C03638=1020.373,204.181,377.085,168.836,50.366,159.543
C03639=1020.379,204.400,377.063,168.838,50.360,159.542
C03640=1020.384,204.618,377.040,168.842,50.355,159.542
C03641=1020.390,204.838,377.018,168.844,50.349,159.541
C03642=1020.396,205.057,376.996,168.848,50.344,159.540
C03643=1020.401,205.276,376.974,168.852,50.339,159.540
C03644=1020.406,205.494,376.951,168.855,50.333,159.539
C03645=1020.412,205.713,376.930,168.858,50.328,159.539
C03646=1020.418,205.961,376.904,168.861,50.322,159.538
C03647=1020.424,206.210,376.879,168.864,50.316,159.537
C03648=1020.431,206.459,376.854,168.868,50.310,159.536
C03649=1020.437,206.707,376.828,168.872,50.304,159.536
C03650=1020.443,206.956,376.803,168.876,50.298,159.535
C03651=1020.449,207.204,376.778,168.879,50.292,159.535
C03652=1020.455,207.453,376.753,168.882,50.287,159.534
C03653=1020.461,207.701,376.727,168.886,50.281,159.533
C03654=1020.466,207.950,376.701,168.890,50.275,159.532
C03655=1020.473,208.198,376.675,168.894,50.269,159.532
C03656=1020.479,208.447,376.650,168.897,50.263,159.531
C03657=1020.485,208.696,376.625,168.900,50.257,159.530
C03658=1020.492,208.944,376.599,168.904,50.251,159.530
C03659=1020.498,209.193,376.574,168.908,50.245,159.529
C03660=1020.504,209.442,376.549,168.912,50.239,159.528
C03661=1020.510,209.690,376.523,168.914,50.233,159.528
C03662=1020.516,209.939,376.497,168.919,50.228,159.527
C03663=1020.522,210.187,376.471,168.922,50.222,159.527
C03664=1020.528,210.436,376.446,168.926,50.216,159.526
C03665=1020.535,210.685,376.421,168.929,50.210,159.525
C03666=1020.540,210.933,376.394,168.933,50.205,159.525
C03667=1020.547,211.182,376.369,168.937,50.199,159.524
C03668=1020.553,211.431,376.343,168.941,50.193,159.524
C03669=1020.559,211.680,376.317,168.944,50.187,159.523
C03670=1020.565,211.928,376.291,168.948,50.182,159.522
C03671=1020.572,212.177,376.266,168.952,50.176,159.522
C03672=1020.577,212.426,376.240,168.954,50.170,159.521
C03673=1020.584,212.674,376.214,168.958,50.164,159.520
C03674=1020.590,212.923,376.188,168.962,50.159,159.520
C03675=1020.596,213.171,376.163,168.966,50.153,159.519
C03676=1020.602,213.420,376.136,168.969,50.147,159.518
C03677=1020.608,213.668,376.111,168.973,50.142,159.518
C03678=1020.614,213.916,376.085,168.977,50.136,159.517
C03679=1020.620,214.165,376.059,168.980,50.130,159.517
C03680=1020.626,214.414,376.034,168.984,50.125,159.516
C03681=1020.633,214.663,376.007,168.988,50.119,159.515
C03682=1020.639,214.912,375.981,168.992,50.114,159.515
C03683=1020.645,215.160,375.955,168.995,50.108,159.514
C03684=1020.651,215.408,375.930,168.999,50.102,159.514
C03685=1020.657,215.657,375.903,169.003,50.097,159.513
C03686=1020.663,215.905,375.878,169.006,50.091,159.512
C03687=1020.670,216.154,375.853,169.010,50.086,159.512
C03688=1020.676,216.403,375.826,169.014,50.080,159.511
C03689=1020.682,216.652,375.800,169.017,50.074,159.511
C03690=1020.689,216.900,375.774,169.021,50.069,159.510
C03691=1020.694,217.149,375.748,169.025,50.063,159.509
C03692=1020.701,217.397,375.722,169.029,50.058,159.509
C03693=1020.707,217.646,375.697,169.032,50.052,159.508
C03694=1020.714,217.894,375.670,169.036,50.047,159.508
C03695=1020.720,218.143,375.644,169.040,50.041,159.507
C03696=1020.726,218.391,375.618,169.044,50.035,159.507
C03697=1020.732,218.640,375.592,169.047,50.030,159.506
C03698=1020.737,218.861,375.569,169.050,50.025,159.506
C03699=1020.743,219.082,375.545,169.053,50.020,159.505
C03700=1020.748,219.304,375.522,169.057,50.015,159.505
C03701=1020.754,219.525,375.498,169.060,50.011,159.504
C03702=1020.759,219.747,375.475,169.063,50.006,159.504
C03703=1020.764,219.968,375.451,169.066,50.001,159.503
C03704=1020.770,220.190,375.429,169.070,49.996,159.503
C03705=1020.775,220.410,375.405,169.073,49.991,159.502
C03706=1020.781,220.659,375.378,169.077,49.986,159.502
C03707=1020.788,220.908,375.353,169.081,49.981,159.501
C03708=1020.794,221.157,375.326,169.084,49.976,159.501
C03709=1020.800,221.405,375.299,169.088,49.970,159.500
C03710=1020.806,221.653,375.273,169.092,49.965,159.499
C03711=1020.812,221.902,375.246,169.096,49.960,159.499
C03712=1020.819,222.151,375.221,169.100,49.954,159.498
C03713=1020.824,222.399,375.194,169.103,49.949,159.498
C03714=1020.830,222.647,375.168,169.107,49.943,159.497
C03715=1020.837,222.896,375.141,169.111,49.938,159.497
C03716=1020.843,223.144,375.115,169.114,49.933,159.496
C03717=1020.849,223.393,375.088,169.118,49.927,159.496
C03718=1020.856,223.642,375.062,169.121,49.922,159.495
C03719=1020.861,223.891,375.036,169.126,49.917,159.495
C03720=1020.868,224.139,375.009,169.130,49.912,159.494
C03721=1020.874,224.387,374.983,169.133,49.907,159.494
C03722=1020.880,224.636,374.956,169.137,49.901,159.493
C03723=1020.887,224.884,374.930,169.141,49.895,159.492
C03724=1020.892,225.132,374.903,169.144,49.890,159.492
C03725=1020.899,225.382,374.876,169.149,49.885,159.491
C03726=1020.905,225.630,374.850,169.152,49.880,159.491
C03727=1020.912,225.879,374.823,169.156,49.875,159.490
C03728=1020.918,226.127,374.797,169.160,49.870,159.490
C03729=1020.924,226.375,374.770,169.163,49.865,159.489
C03730=1020.930,226.624,374.743,169.167,49.859,159.489
C03731=1020.937,226.872,374.717,169.171,49.853,159.488
C03732=1020.943,227.120,374.691,169.175,49.849,159.488
C03733=1020.949,227.370,374.664,169.179,49.844,159.488
C03734=1020.955,227.618,374.637,169.182,49.839,159.487
C03735=1020.961,227.866,374.610,169.187,49.834,159.487
C03736=1020.967,228.115,374.583,169.190,49.829,159.486
C03737=1020.973,228.364,374.557,169.194,49.824,159.486
C03738=1020.980,228.612,374.530,169.197,49.819,159.485
C03739=1020.986,228.860,374.503,169.202,49.813,159.485
C03740=1020.992,229.109,374.476,169.206,49.808,159.484
C03741=1020.998,229.358,374.449,169.209,49.803,159.483
C03742=1021.004,229.606,374.423,169.213,49.798,159.483
C03743=1021.010,229.855,374.396,169.216,49.793,159.482
C03744=1021.016,230.103,374.368,169.221,49.788,159.482
C03745=1021.022,230.351,374.342,169.224,49.783,159.482
C03746=1021.028,230.600,374.315,169.228,49.778,159.481
C03747=1021.034,230.848,374.287,169.232,49.773,159.481
C03748=1021.041,231.097,374.260,169.236,49.768,159.480
C03749=1021.047,231.345,374.233,169.241,49.763,159.480
C03750=1021.053,231.594,374.206,169.244,49.758,159.479
C03751=1021.059,231.842,374.179,169.248,49.753,159.479
C03752=1021.065,232.091,374.152,169.251,49.748,159.478
C03753=1021.072,232.339,374.125,169.256,49.744,159.478
C03754=1021.077,232.587,374.098,169.259,49.739,159.478
C03755=1021.084,232.836,374.071,169.263,49.733,159.477
C03756=1021.090,233.084,374.044,169.266,49.728,159.477
C03757=1021.096,233.333,374.017,169.271,49.724,159.476
C03758=1021.101,233.550,373.993,169.275,49.720,159.476
C03759=1021.107,233.767,373.969,169.277,49.716,159.476
C03760=1021.113,233.985,373.945,169.280,49.711,159.475
C03761=1021.117,234.202,373.922,169.284,49.706,159.475
C03762=1021.123,234.419,373.897,169.288,49.702,159.474
C03763=1021.129,234.637,373.874,169.291,49.698,159.474
C03764=1021.134,234.854,373.851,169.295,49.694,159.474
C03765=1021.140,235.071,373.826,169.297,49.690,159.473
C03766=1021.145,235.320,373.800,169.302,49.684,159.473
C03767=1021.152,235.568,373.772,169.306,49.680,159.472
C03768=1021.158,235.817,373.745,169.309,49.675,159.472
C03769=1021.164,236.065,373.717,169.314,49.670,159.472
C03770=1021.171,236.314,373.690,169.317,49.665,159.471
C03771=1021.177,236.562,373.663,169.322,49.661,159.471
C03772=1021.183,236.811,373.636,169.325,49.656,159.470
C03773=1021.189,237.059,373.609,169.329,49.651,159.470
C03774=1021.195,237.307,373.580,169.333,49.646,159.469
C03775=1021.202,237.556,373.553,169.337,49.641,159.469
C03776=1021.208,237.804,373.526,169.341,49.637,159.469
C03777=1021.214,238.053,373.499,169.345,49.632,159.468
C03778=1021.220,238.301,373.472,169.349,49.627,159.468
C03779=1021.227,238.549,373.444,169.353,49.622,159.467
C03780=1021.233,238.798,373.417,169.356,49.618,159.467
C03781=1021.239,239.046,373.389,169.361,49.613,159.466
C03782=1021.246,239.295,373.362,169.364,49.609,159.466
C03783=1021.251,239.543,373.334,169.369,49.604,159.466
C03784=1021.258,239.792,373.307,169.372,49.599,159.465
C03785=1021.264,240.040,373.278,169.377,49.594,159.465
C03786=1021.270,240.288,373.251,169.380,49.590,159.465
C03787=1021.276,240.537,373.223,169.385,49.585,159.464
C03788=1021.282,240.785,373.195,169.388,49.581,159.464
C03789=1021.289,241.033,373.168,169.393,49.576,159.464
C03790=1021.295,241.282,373.141,169.396,49.571,159.463
C03791=1021.301,241.531,373.112,169.400,49.567,159.463
C03792=1021.307,241.779,373.085,169.404,49.562,159.462
C03793=1021.313,242.027,373.057,169.408,49.558,159.462
C03794=1021.320,242.276,373.029,169.412,49.553,159.462
C03795=1021.326,242.524,373.002,169.416,49.549,159.461
C03796=1021.332,242.772,372.973,169.420,49.544,159.461
C03797=1021.338,243.021,372.945,169.424,49.540,159.461
C03798=1021.344,243.268,372.918,169.429,49.535,159.460
C03799=1021.350,243.517,372.890,169.432,49.530,159.460
C03800=1021.357,243.766,372.862,169.436,49.526,159.460
C03801=1021.362,244.014,372.834,169.440,49.522,159.459
C03802=1021.368,244.262,372.806,169.444,49.517,159.459
C03803=1021.375,244.511,372.778,169.448,49.513,159.459
C03804=1021.381,244.760,372.750,169.452,49.509,159.458
C03805=1021.386,245.008,372.722,169.456,49.504,159.458
C03806=1021.393,245.256,372.693,169.460,49.500,159.458
C03807=1021.399,245.504,372.665,169.464,49.496,159.457
C03808=1021.404,245.752,372.637,169.468,49.491,159.457
C03809=1021.411,246.001,372.609,169.472,49.487,159.457
C03810=1021.417,246.250,372.581,169.477,49.482,159.456
C03811=1021.423,246.498,372.552,169.480,49.478,159.456
C03812=1021.429,246.745,372.525,169.485,49.473,159.456
C03813=1021.435,246.994,372.496,169.488,49.469,159.455
C03814=1021.441,247.243,372.468,169.492,49.465,159.455
C03815=1021.448,247.491,372.439,169.497,49.460,159.455
C03816=1021.454,247.740,372.411,169.500,49.456,159.454
C03817=1021.460,247.988,372.383,169.505,49.452,159.454
C03818=1021.465,248.202,372.359,169.508,49.448,159.454
C03819=1021.470,248.416,372.335,169.511,49.444,159.453
C03820=1021.476,248.630,372.310,169.515,49.441,159.453
C03821=1021.482,248.844,372.286,169.518,49.437,159.453
C03822=1021.486,249.058,372.261,169.522,49.433,159.453
C03823=1021.492,249.273,372.237,169.526,49.430,159.452
C03824=1021.497,249.487,372.213,169.529,49.426,159.452
C03825=1021.503,249.701,372.188,169.532,49.422,159.452
C03826=1021.509,249.950,372.160,169.536,49.419,159.452
C03827=1021.515,250.197,372.131,169.541,49.414,159.451
C03828=1021.521,250.445,372.103,169.545,49.410,159.451
C03829=1021.527,250.694,372.075,169.549,49.405,159.451
C03830=1021.533,250.942,372.046,169.553,49.401,159.450
C03831=1021.540,251.191,372.018,169.558,49.396,159.450
C03832=1021.546,251.439,371.989,169.562,49.393,159.450
C03833=1021.552,251.688,371.961,169.565,49.389,159.450
C03834=1021.559,251.936,371.933,169.570,49.384,159.449
C03835=1021.565,252.184,371.904,169.573,49.380,159.449
C03836=1021.571,252.433,371.876,169.578,49.375,159.449
C03837=1021.578,252.680,371.848,169.582,49.372,159.449
C03838=1021.584,252.929,371.819,169.587,49.367,159.448
C03839=1021.590,253.177,371.790,169.590,49.363,159.448
C03840=1021.596,253.425,371.763,169.594,49.359,159.448
C03841=1021.603,253.674,371.733,169.599,49.355,159.447
C03842=1021.609,253.922,371.705,169.602,49.351,159.447
C03843=1021.616,254.170,371.677,169.607,49.346,159.447
C03844=1021.622,254.418,371.648,169.611,49.343,159.447
C03845=1021.628,254.667,371.619,169.616,49.338,159.446
C03846=1021.634,254.915,371.590,169.619,49.334,159.446
C03847=1021.641,255.164,371.563,169.624,49.329,159.446
C03848=1021.647,255.412,371.534,169.628,49.326,159.446
C03849=1021.653,255.660,371.504,169.631,49.322,159.445
C03850=1021.660,255.908,371.477,169.636,49.318,159.445
C03851=1021.666,256.156,371.448,169.640,49.314,159.445
C03852=1021.672,256.405,371.419,169.645,49.309,159.444
C03853=1021.679,256.653,371.391,169.649,49.306,159.444
C03854=1021.685,256.901,371.362,169.653,49.301,159.444
C03855=1021.692,257.151,371.333,169.657,49.297,159.444
C03856=1021.699,257.398,371.305,169.662,49.293,159.444
C03857=1021.705,257.647,371.276,169.666,49.289,159.443
C03858=1021.711,257.895,371.247,169.670,49.285,159.443
C03859=1021.717,258.143,371.218,169.674,49.281,159.443
C03860=1021.724,258.391,371.190,169.678,49.277,159.443
C03861=1021.731,258.639,371.161,169.683,49.273,159.442
C03862=1021.737,258.887,371.132,169.687,49.269,159.442
C03863=1021.744,259.136,371.104,169.691,49.265,159.442
C03864=1021.750,259.384,371.075,169.695,49.260,159.442
C03865=1021.757,259.633,371.046,169.700,49.256,159.441
C03866=1021.764,259.881,371.017,169.704,49.252,159.441
C03867=1021.770,260.129,370.988,169.709,49.248,159.441
C03868=1021.776,260.377,370.959,169.713,49.245,159.441
C03869=1021.782,260.625,370.930,169.716,49.241,159.440
C03870=1021.789,260.873,370.901,169.721,49.237,159.440
C03871=1021.795,261.121,370.872,169.725,49.233,159.440
C03872=1021.801,261.369,370.843,169.730,49.229,159.440
C03873=1021.807,261.618,370.814,169.734,49.225,159.440
C03874=1021.813,261.867,370.784,169.738,49.222,159.440
C03875=1021.820,262.115,370.755,169.743,49.218,159.439
C03876=1021.826,262.363,370.726,169.746,49.214,159.439
C03877=1021.832,262.611,370.697,169.750,49.210,159.439
C03878=1021.838,262.824,370.672,169.754,49.207,159.439
C03879=1021.843,263.038,370.646,169.759,49.204,159.439
C03880=1021.849,263.251,370.621,169.762,49.200,159.439
C03881=1021.854,263.464,370.596,169.766,49.197,159.438
C03882=1021.860,263.678,370.571,169.770,49.193,159.438
C03883=1021.865,263.891,370.546,169.773,49.191,159.438
C03884=1021.870,264.104,370.521,169.777,49.187,159.438
C03885=1021.876,264.318,370.495,169.781,49.184,159.438
C03886=1021.882,264.566,370.466,169.785,49.180,159.438
C03887=1021.888,264.814,370.437,169.789,49.177,159.437
C03888=1021.895,265.062,370.407,169.794,49.173,159.437
C03889=1021.901,265.310,370.378,169.798,49.169,159.437
C03890=1021.908,265.559,370.348,169.803,49.165,159.437
C03891=1021.914,265.807,370.319,169.807,49.162,159.437
C03892=1021.920,266.055,370.289,169.810,49.158,159.437
C03893=1021.926,266.303,370.260,169.815,49.154,159.436
C03894=1021.933,266.552,370.231,169.819,49.150,159.436
C03895=1021.940,266.799,370.201,169.823,49.147,159.436
C03896=1021.945,267.048,370.171,169.828,49.143,159.436
C03897=1021.952,267.296,370.141,169.832,49.139,159.436
C03898=1021.958,267.544,370.112,169.837,49.136,159.436
C03899=1021.965,267.792,370.083,169.841,49.132,159.436
C03900=1021.971,268.040,370.053,169.846,49.129,159.436
C03901=1021.977,268.289,370.023,169.851,49.125,159.435
C03902=1021.984,268.536,369.993,169.855,49.122,159.435
C03903=1021.989,268.785,369.964,169.860,49.118,159.435
C03904=1021.997,269.033,369.934,169.864,49.114,159.435
C03905=1022.003,269.281,369.905,169.868,49.111,159.435
C03906=1022.009,269.528,369.875,169.873,49.107,159.435
C03907=1022.016,269.778,369.845,169.877,49.104,159.435
C03908=1022.022,270.025,369.815,169.882,49.100,159.434
C03909=1022.028,270.273,369.785,169.886,49.097,159.435
C03910=1022.035,270.522,369.755,169.890,49.093,159.434
C03911=1022.041,270.770,369.725,169.895,49.089,159.434
C03912=1022.047,271.017,369.695,169.899,49.086,159.434
C03913=1022.054,271.266,369.666,169.903,49.082,159.434
C03914=1022.060,271.514,369.635,169.908,49.079,159.434
C03915=1022.067,271.762,369.605,169.912,49.076,159.434
C03916=1022.072,272.010,369.576,169.917,49.072,159.434
C03917=1022.079,272.258,369.546,169.921,49.068,159.434
C03918=1022.085,272.506,369.515,169.926,49.066,159.434
C03919=1022.092,272.754,369.486,169.931,49.062,159.433
C03920=1022.098,273.003,369.456,169.935,49.058,159.433
C03921=1022.105,273.251,369.426,169.939,49.055,159.433
C03922=1022.110,273.498,369.395,169.944,49.051,159.433
C03923=1022.118,273.747,369.365,169.948,49.048,159.433
C03924=1022.123,273.995,369.335,169.953,49.045,159.433
C03925=1022.131,274.243,369.305,169.957,49.041,159.433
C03926=1022.136,274.491,369.275,169.961,49.038,159.433
C03927=1022.143,274.739,369.245,169.967,49.035,159.433
C03928=1022.149,274.987,369.215,169.971,49.031,159.433
C03929=1022.156,275.236,369.184,169.975,49.028,159.433
C03930=1022.162,275.483,369.154,169.980,49.024,159.433
C03931=1022.169,275.732,369.124,169.984,49.021,159.433
C03932=1022.175,275.979,369.094,169.989,49.018,159.433
C03933=1022.181,276.228,369.063,169.993,49.014,159.432
C03934=1022.188,276.475,369.033,169.998,49.011,159.432
C03935=1022.194,276.724,369.003,170.003,49.007,159.432
C03936=1022.201,276.971,368.973,170.007,49.005,159.432
C03937=1022.207,277.220,368.942,170.012,49.001,159.432
C03938=1022.213,277.435,368.915,170.015,48.998,159.432
C03939=1022.218,277.651,368.889,170.020,48.995,159.432
C03940=1022.223,277.867,368.862,170.024,48.993,159.432
C03941=1022.230,278.082,368.836,170.027,48.990,159.432
C03942=1022.235,278.298,368.809,170.032,48.987,159.432
C03943=1022.240,278.514,368.783,170.036,48.984,159.432
C03944=1022.245,278.729,368.756,170.039,48.982,159.432
C03945=1022.251,278.945,368.729,170.044,48.979,159.432
C03946=1022.258,279.192,368.699,170.048,48.976,159.432
C03947=1022.264,279.440,368.668,170.053,48.972,159.432
C03948=1022.271,279.689,368.638,170.057,48.969,159.432
C03949=1022.277,279.937,368.607,170.062,48.966,159.432
C03950=1022.283,280.185,368.576,170.067,48.963,159.432
C03951=1022.290,280.432,368.546,170.071,48.960,159.432
C03952=1022.296,280.681,368.515,170.076,48.957,159.432
C03953=1022.303,280.929,368.485,170.081,48.954,159.432
C03954=1022.309,281.176,368.453,170.085,48.951,159.432
C03955=1022.315,281.425,368.423,170.090,48.947,159.432
C03956=1022.322,281.673,368.393,170.094,48.944,159.432
C03957=1022.328,281.920,368.362,170.099,48.941,159.432
C03958=1022.335,282.169,368.331,170.104,48.938,159.432
C03959=1022.342,282.417,368.299,170.108,48.935,159.432
C03960=1022.347,282.665,368.269,170.113,48.932,159.432
C03961=1022.355,282.913,368.239,170.118,48.929,159.432
C03962=1022.361,283.161,368.208,170.122,48.926,159.432
C03963=1022.368,283.409,368.177,170.127,48.923,159.432
C03964=1022.374,283.656,368.146,170.132,48.920,159.432
C03965=1022.380,283.905,368.115,170.137,48.917,159.432
C03966=1022.387,284.153,368.084,170.141,48.913,159.432
C03967=1022.394,284.400,368.054,170.146,48.910,159.432
C03968=1022.400,284.648,368.022,170.151,48.907,159.432
C03969=1022.407,284.897,367.992,170.155,48.904,159.432
C03970=1022.413,285.145,367.960,170.161,48.901,159.432
C03971=1022.420,285.393,367.929,170.165,48.898,159.432
C03972=1022.426,285.640,367.898,170.170,48.895,159.432
C03973=1022.433,285.888,367.867,170.175,48.892,159.432
C03974=1022.439,286.136,367.836,170.179,48.889,159.432
C03975=1022.446,286.385,367.805,170.184,48.886,159.432
C03976=1022.452,286.632,367.774,170.189,48.883,159.432
C03977=1022.459,286.880,367.742,170.194,48.880,159.432
C03978=1022.465,287.128,367.712,170.199,48.878,159.433
C03979=1022.472,287.376,367.680,170.203,48.875,159.433
C03980=1022.479,287.624,367.649,170.208,48.872,159.433
C03981=1022.485,287.871,367.618,170.213,48.869,159.433
C03982=1022.491,288.119,367.586,170.218,48.866,159.433
C03983=1022.498,288.368,367.556,170.222,48.863,159.433
C03984=1022.505,288.616,367.524,170.227,48.860,159.433
C03985=1022.511,288.864,367.492,170.232,48.858,159.433
C03986=1022.517,289.112,367.461,170.237,48.855,159.433
C03987=1022.524,289.360,367.429,170.242,48.852,159.433
C03988=1022.530,289.607,367.398,170.246,48.849,159.433
C03989=1022.537,289.855,367.367,170.251,48.846,159.433
C03990=1022.544,290.103,367.335,170.257,48.844,159.433
C03991=1022.550,290.351,367.304,170.261,48.841,159.433
C03992=1022.557,290.599,367.272,170.266,48.838,159.434
C03993=1022.563,290.847,367.240,170.271,48.835,159.434
C03994=1022.570,291.095,367.209,170.276,48.832,159.434
C03995=1022.576,291.343,367.178,170.281,48.829,159.434
C03996=1022.583,291.591,367.146,170.285,48.827,159.434
C03997=1022.590,291.838,367.115,170.291,48.824,159.434
C03998=1022.595,292.060,367.086,170.295,48.821,159.434
C03999=1022.601,292.281,367.058,170.299,48.819,159.434
C04000=1022.607,292.504,367.029,170.303,48.817,159.434
C04001=1022.614,292.725,367.001,170.308,48.814,159.434
C04002=1022.619,292.947,366.973,170.312,48.812,159.435
C04003=1022.625,293.168,366.945,170.317,48.809,159.435
C04004=1022.631,293.390,366.916,170.321,48.807,159.435
C04005=1022.637,293.613,366.888,170.326,48.805,159.435
C04006=1022.643,293.860,366.856,170.330,48.802,159.435
C04007=1022.649,294.109,366.824,170.335,48.800,159.435
C04008=1022.656,294.356,366.792,170.341,48.797,159.435
C04009=1022.662,294.604,366.760,170.345,48.795,159.435
C04010=1022.669,294.852,366.728,170.350,48.792,159.436
C04011=1022.675,295.100,366.695,170.355,48.789,159.436
C04012=1022.681,295.348,366.663,170.360,48.787,159.436
C04013=1022.688,295.595,366.631,170.366,48.785,159.436
C04014=1022.694,295.843,366.599,170.370,48.782,159.436
C04015=1022.701,296.090,366.567,170.375,48.780,159.436
C04016=1022.707,296.339,366.535,170.380,48.777,159.437
C04017=1022.714,296.586,366.502,170.385,48.774,159.437
C04018=1022.720,296.834,366.471,170.390,48.772,159.437
C04019=1022.727,297.082,366.438,170.395,48.769,159.437
C04020=1022.733,297.330,366.407,170.400,48.767,159.437
C04021=1022.740,297.577,366.374,170.405,48.764,159.437
C04022=1022.746,297.825,366.341,170.410,48.762,159.438
C04023=1022.753,298.073,366.310,170.416,48.759,159.438
C04024=1022.759,298.320,366.277,170.420,48.757,159.438
C04025=1022.766,298.569,366.245,170.425,48.754,159.438
C04026=1022.773,298.817,366.212,170.430,48.752,159.438
C04027=1022.779,299.064,366.180,170.435,48.750,159.439
C04028=1022.786,299.312,366.148,170.441,48.747,159.439
C04029=1022.792,299.560,366.116,170.445,48.745,159.439
C04030=1022.799,299.807,366.083,170.451,48.743,159.439
C04031=1022.805,300.055,366.051,170.456,48.740,159.440
C04032=1022.812,300.303,366.018,170.461,48.737,159.440
C04033=1022.819,300.551,365.986,170.466,48.735,159.440
C04034=1022.825,300.798,365.953,170.470,48.733,159.440
C04035=1022.832,301.046,365.921,170.476,48.730,159.440
C04036=1022.839,301.295,365.889,170.481,48.728,159.440
C04037=1022.845,301.542,365.856,170.487,48.726,159.441
C04038=1022.852,301.789,365.824,170.491,48.724,159.441
C04039=1022.858,302.037,365.791,170.497,48.721,159.441
C04040=1022.865,302.285,365.758,170.502,48.719,159.441
C04041=1022.872,302.533,365.726,170.507,48.716,159.442
C04042=1022.879,302.780,365.693,170.512,48.714,159.442
C04043=1022.886,303.027,365.661,170.518,48.712,159.442
C04044=1022.892,303.276,365.629,170.522,48.709,159.442
C04045=1022.898,303.524,365.596,170.528,48.707,159.443
C04046=1022.905,303.771,365.564,170.533,48.705,159.443
C04047=1022.912,304.020,365.531,170.539,48.702,159.443
C04048=1022.919,304.267,365.498,170.543,48.700,159.443
C04049=1022.926,304.514,365.466,170.549,48.698,159.443
C04050=1022.933,304.763,365.433,170.554,48.695,159.444
C04051=1022.940,305.010,365.400,170.559,48.693,159.444
C04052=1022.947,305.258,365.367,170.564,48.691,159.444
C04053=1022.953,305.505,365.334,170.570,48.689,159.445
C04054=1022.960,305.753,365.302,170.575,48.687,159.445
C04055=1022.967,306.001,365.269,170.580,48.684,159.445
C04056=1022.973,306.248,365.236,170.585,48.682,159.445
C04057=1022.981,306.496,365.203,170.591,48.680,159.445
C04058=1022.987,306.727,365.173,170.596,48.678,159.446
C04059=1022.993,306.958,365.142,170.601,48.676,159.446
C04060=1023.000,307.188,365.111,170.605,48.674,159.446
C04061=1023.006,307.418,365.081,170.610,48.671,159.446
C04062=1023.013,307.648,365.051,170.615,48.670,159.447
C04063=1023.019,307.879,365.021,170.621,48.667,159.447
C04064=1023.025,308.109,364.989,170.625,48.665,159.447
C04065=1023.032,308.340,364.959,170.630,48.664,159.448
C04066=1023.039,308.588,364.926,170.636,48.661,159.448
C04067=1023.046,308.835,364.894,170.641,48.659,159.448
C04068=1023.053,309.083,364.860,170.647,48.657,159.449
C04069=1023.060,309.330,364.828,170.651,48.655,159.449
C04070=1023.067,309.578,364.794,170.657,48.652,159.449
C04071=1023.073,309.825,364.761,170.662,48.651,159.449
C04072=1023.081,310.073,364.728,170.668,48.648,159.450
C04073=1023.088,310.321,364.695,170.674,48.646,159.450
C04074=1023.094,310.569,364.662,170.679,48.644,159.450
C04075=1023.102,310.816,364.628,170.684,48.643,159.451
C04076=1023.108,311.064,364.594,170.689,48.640,159.451
C04077=1023.114,311.312,364.561,170.694,48.639,159.451
C04078=1023.121,311.559,364.527,170.700,48.637,159.452
C04079=1023.128,311.807,364.494,170.705,48.635,159.452
C04080=1023.134,312.054,364.460,170.711,48.633,159.452
C04081=1023.141,312.302,364.426,170.716,48.631,159.453
C04082=1023.148,312.549,364.393,170.722,48.629,159.453
C04083=1023.154,312.797,364.359,170.727,48.627,159.453
C04084=1023.161,313.045,364.325,170.733,48.626,159.454
C04085=1023.168,313.292,364.292,170.738,48.623,159.454
C04086=1023.175,313.540,364.258,170.744,48.622,159.454
C04087=1023.181,313.787,364.224,170.750,48.620,159.455
C04088=1023.188,314.035,364.190,170.755,48.618,159.455
C04089=1023.195,314.283,364.156,170.761,48.616,159.456
C04090=1023.202,314.530,364.123,170.766,48.614,159.456
C04091=1023.208,314.778,364.089,170.772,48.612,159.456
C04092=1023.215,315.025,364.055,170.777,48.611,159.457
C04093=1023.222,315.272,364.021,170.783,48.609,159.457
C04094=1023.228,315.520,363.987,170.788,48.607,159.458
C04095=1023.236,315.768,363.953,170.794,48.605,159.458
C04096=1023.243,316.016,363.919,170.798,48.603,159.458
C04097=1023.249,316.263,363.886,170.804,48.601,159.459
C04098=1023.256,316.511,363.851,170.810,48.600,159.459
C04099=1023.263,316.758,363.818,170.815,48.598,159.460
C04100=1023.270,317.006,363.784,170.822,48.596,159.460
C04101=1023.276,317.253,363.750,170.827,48.595,159.460
C04102=1023.283,317.501,363.716,170.833,48.593,159.461
C04103=1023.290,317.749,363.682,170.838,48.591,159.461
C04104=1023.298,317.996,363.648,170.844,48.589,159.462
C04105=1023.304,318.244,363.614,170.850,48.588,159.462
C04106=1023.312,318.491,363.579,170.855,48.586,159.462
C04107=1023.318,318.738,363.546,170.861,48.584,159.463
C04108=1023.325,318.986,363.511,170.866,48.583,159.463
C04109=1023.332,319.234,363.478,170.872,48.581,159.464
C04110=1023.339,319.482,363.444,170.878,48.579,159.464
C04111=1023.346,319.729,363.409,170.883,48.577,159.465
C04112=1023.353,319.977,363.375,170.889,48.576,159.465
C04113=1023.360,320.224,363.341,170.895,48.574,159.466
C04114=1023.367,320.472,363.307,170.900,48.573,159.466
C04115=1023.374,320.719,363.272,170.906,48.571,159.466
C04116=1023.381,320.967,363.238,170.911,48.569,159.467
C04117=1023.389,321.215,363.204,170.917,48.568,159.467
C04118=1023.395,321.447,363.172,170.922,48.566,159.468
C04119=1023.402,321.680,363.140,170.929,48.565,159.468
C04120=1023.408,321.914,363.107,170.934,48.563,159.469
C04121=1023.414,322.146,363.075,170.939,48.562,159.469
C04122=1023.421,322.379,363.042,170.945,48.560,159.469
C04123=1023.428,322.613,363.010,170.950,48.558,159.470
C04124=1023.436,322.846,362.978,170.955,48.557,159.470
C04125=1023.442,323.078,362.946,170.961,48.556,159.471
C04126=1023.448,323.326,362.911,170.966,48.554,159.471
C04127=1023.456,323.574,362.876,170.973,48.553,159.472
C04128=1023.464,323.821,362.842,170.979,48.551,159.472
C04129=1023.470,324.069,362.807,170.985,48.549,159.473
C04130=1023.478,324.316,362.773,170.990,48.548,159.473
C04131=1023.485,324.563,362.738,170.996,48.546,159.474
C04132=1023.492,324.811,362.704,171.002,48.545,159.474
C04133=1023.499,325.058,362.669,171.008,48.544,159.475
C04134=1023.507,325.307,362.635,171.014,48.542,159.475
C04135=1023.514,325.554,362.600,171.020,48.540,159.476
C04136=1023.521,325.801,362.566,171.026,48.539,159.476
C04137=1023.528,326.049,362.532,171.031,48.537,159.477
C04138=1023.535,326.296,362.497,171.038,48.536,159.477
C04139=1023.543,326.544,362.462,171.044,48.534,159.478
C04140=1023.551,326.791,362.427,171.049,48.533,159.478
C04141=1023.558,327.038,362.392,171.055,48.531,159.479
C04142=1023.565,327.286,362.358,171.061,48.530,159.479
C04143=1023.572,327.533,362.323,171.068,48.529,159.480
C04144=1023.579,327.781,362.288,171.073,48.527,159.480
C04145=1023.586,328.028,362.252,171.079,48.526,159.481
C04146=1023.594,328.275,362.217,171.086,48.525,159.482
C04147=1023.600,328.522,362.182,171.091,48.523,159.482
C04148=1023.607,328.770,362.147,171.097,48.522,159.483
C04149=1023.614,329.018,362.111,171.103,48.521,159.483
C04150=1023.622,329.265,362.077,171.110,48.520,159.484
C04151=1023.629,329.512,362.042,171.115,48.519,159.485
C04152=1023.636,329.760,362.006,171.121,48.517,159.485
C04153=1023.643,330.008,361.971,171.127,48.516,159.486
C04154=1023.650,330.254,361.935,171.133,48.515,159.486
C04155=1023.658,330.502,361.900,171.139,48.514,159.487
C04156=1023.665,330.750,361.865,171.146,48.512,159.487
C04157=1023.672,330.997,361.830,171.152,48.511,159.488
C04158=1023.679,331.245,361.795,171.158,48.510,159.489
C04159=1023.686,331.492,361.759,171.163,48.508,159.489
C04160=1023.694,331.739,361.724,171.170,48.507,159.490
C04161=1023.701,331.987,361.689,171.176,48.506,159.490
C04162=1023.708,332.234,361.653,171.182,48.505,159.491
C04163=1023.715,332.482,361.617,171.188,48.504,159.492
C04164=1023.723,332.729,361.583,171.194,48.503,159.492
C04165=1023.731,332.976,361.547,171.201,48.501,159.493
C04166=1023.737,333.224,361.511,171.207,48.500,159.494
C04167=1023.745,333.471,361.475,171.213,48.499,159.494
C04168=1023.752,333.718,361.440,171.219,48.499,159.495
C04169=1023.759,333.965,361.404,171.225,48.497,159.496
C04170=1023.766,334.213,361.369,171.232,48.496,159.496
C04171=1023.773,334.460,361.333,171.238,48.495,159.497
C04172=1023.781,334.707,361.297,171.244,48.494,159.497
C04173=1023.788,334.955,361.261,171.250,48.493,159.498
C04174=1023.795,335.202,361.225,171.257,48.492,159.499
C04175=1023.803,335.450,361.189,171.263,48.491,159.499
C04176=1023.810,335.697,361.154,171.269,48.490,159.500
C04177=1023.818,335.944,361.118,171.276,48.489,159.501
C04178=1023.824,336.175,361.084,171.281,48.488,159.502
C04179=1023.831,336.406,361.050,171.287,48.487,159.502
C04180=1023.838,336.637,361.017,171.293,48.486,159.503
C04181=1023.844,336.867,360.984,171.299,48.485,159.503
C04182=1023.852,337.098,360.950,171.305,48.485,159.504
C04183=1023.858,337.329,360.916,171.311,48.484,159.505
C04184=1023.865,337.560,360.883,171.317,48.483,159.505
C04185=1023.872,337.790,360.849,171.322,48.482,159.506
C04186=1023.880,338.037,360.813,171.329,48.481,159.507
C04187=1023.887,338.285,360.778,171.336,48.480,159.507
C04188=1023.894,338.533,360.741,171.342,48.479,159.508
C04189=1023.901,338.780,360.705,171.349,48.478,159.509
C04190=1023.908,339.027,360.669,171.354,48.478,159.510
C04191=1023.916,339.274,360.633,171.361,48.476,159.510
C04192=1023.924,339.522,360.596,171.367,48.476,159.511
C04193=1023.932,339.769,360.560,171.374,48.475,159.512
C04194=1023.939,340.016,360.524,171.380,48.474,159.512
C04195=1023.947,340.263,360.487,171.387,48.473,159.513
C04196=1023.954,340.510,360.451,171.394,48.472,159.514
C04197=1023.961,340.758,360.414,171.400,48.472,159.515
C04198=1023.968,341.005,360.378,171.407,48.470,159.515
C04199=1023.976,341.252,360.341,171.413,48.470,159.516
C04200=1023.983,341.499,360.305,171.419,48.469,159.517
C04201=1023.991,341.747,360.269,171.425,48.468,159.518
C04202=1023.999,341.994,360.232,171.432,48.468,159.518
C04203=1024.006,342.241,360.195,171.439,48.467,159.519
C04204=1024.013,342.488,360.159,171.446,48.466,159.520
C04205=1024.021,342.735,360.122,171.452,48.466,159.521
C04206=1024.028,342.983,360.085,171.459,48.465,159.522
C04207=1024.035,343.230,360.049,171.465,48.464,159.522
C04208=1024.043,343.477,360.012,171.472,48.463,159.523
C04209=1024.050,343.725,359.975,171.479,48.463,159.524
C04210=1024.058,343.971,359.938,171.486,48.462,159.525
C04211=1024.065,344.219,359.901,171.492,48.462,159.526
C04212=1024.073,344.466,359.865,171.499,48.461,159.526
C04213=1024.080,344.713,359.829,171.506,48.460,159.527
C04214=1024.088,344.960,359.791,171.512,48.460,159.528
C04215=1024.096,345.207,359.754,171.519,48.459,159.529
C04216=1024.103,345.454,359.717,171.526,48.459,159.530
C04217=1024.110,345.701,359.680,171.533,48.458,159.531
C04218=1024.118,345.948,359.644,171.539,48.457,159.531
C04219=1024.126,346.197,359.606,171.546,48.457,159.532
C04220=1024.134,346.443,359.569,171.553,48.456,159.533
C04221=1024.141,346.690,359.532,171.559,48.456,159.534
C04222=1024.149,346.937,359.495,171.566,48.455,159.535
C04223=1024.157,347.185,359.459,171.573,48.454,159.536
C04224=1024.164,347.432,359.421,171.579,48.454,159.536
C04225=1024.172,347.679,359.384,171.587,48.454,159.537
C04226=1024.179,347.926,359.347,171.593,48.453,159.538
C04227=1024.187,348.173,359.310,171.600,48.452,159.539
C04228=1024.195,348.420,359.272,171.607,48.452,159.540
C04229=1024.202,348.667,359.235,171.614,48.452,159.541
C04230=1024.210,348.914,359.198,171.620,48.451,159.542
C04231=1024.218,349.162,359.160,171.627,48.451,159.543
C04232=1024.226,349.408,359.123,171.634,48.451,159.544
C04233=1024.233,349.656,359.086,171.641,48.450,159.544
C04234=1024.240,349.903,359.048,171.648,48.449,159.545
C04235=1024.248,350.149,359.010,171.655,48.449,159.546
C04236=1024.256,350.397,358.972,171.661,48.449,159.547
C04237=1024.264,350.644,358.935,171.668,48.449,159.548
C04238=1024.270,350.873,358.900,171.675,48.448,159.549
C04239=1024.278,351.102,358.865,171.682,48.448,159.550
C04240=1024.286,351.332,358.830,171.688,48.448,159.551
C04241=1024.292,351.561,358.796,171.695,48.447,159.551
C04242=1024.299,351.790,358.760,171.701,48.447,159.552
C04243=1024.306,352.019,358.726,171.708,48.447,159.553
C04244=1024.314,352.249,358.691,171.714,48.446,159.554
C04245=1024.322,352.477,358.656,171.721,48.446,159.555
C04246=1024.329,352.724,358.618,171.728,48.446,159.556
C04247=1024.337,352.972,358.580,171.735,48.446,159.557
C04248=1024.345,353.218,358.543,171.742,48.446,159.558
C04249=1024.352,353.465,358.505,171.750,48.445,159.559
C04250=1024.360,353.713,358.467,171.757,48.445,159.560
C04251=1024.369,353.959,358.429,171.764,48.445,159.561
C04252=1024.376,354.207,358.391,171.770,48.444,159.562
C04253=1024.384,354.453,358.353,171.778,48.444,159.563
C04254=1024.391,354.701,358.315,171.785,48.444,159.564
C04255=1024.399,354.948,358.277,171.793,48.444,159.565
C04256=1024.408,355.194,358.239,171.800,48.444,159.566
C04257=1024.415,355.442,358.201,171.807,48.444,159.567
C04258=1024.423,355.688,358.163,171.813,48.443,159.568
C04259=1024.431,355.936,358.124,171.820,48.443,159.569
C04260=1024.439,356.182,358.086,171.829,48.443,159.570
C04261=1024.447,356.430,358.048,171.836,48.443,159.571
C04262=1024.454,356.676,358.010,171.843,48.443,159.572
C04263=1024.463,356.923,357.972,171.850,48.443,159.573
C04264=1024.471,357.170,357.934,171.858,48.443,159.574
C04265=1024.479,357.417,357.895,171.865,48.443,159.575
C04266=1024.486,357.664,357.857,171.872,48.443,159.576
C04267=1024.494,357.911,357.818,171.879,48.443,159.577
C04268=1024.503,358.158,357.780,171.887,48.443,159.578
C04269=1024.510,358.404,357.741,171.894,48.443,159.579
C04270=1024.518,358.652,357.703,171.901,48.443,159.580
C04271=1024.526,358.899,357.664,171.909,48.442,159.581
C04272=1024.534,359.145,357.626,171.916,48.442,159.582
C04273=1024.542,359.393,357.587,171.924,48.442,159.583
C04274=1024.550,359.640,357.549,171.931,48.443,159.585
C04275=1024.559,359.885,357.510,171.939,48.443,159.586
C04276=1024.567,360.133,357.472,171.946,48.443,159.587
C04277=1024.574,360.380,357.433,171.953,48.443,159.588
C04278=1024.582,360.627,357.394,171.961,48.443,159.589
C04279=1024.590,360.873,357.355,171.969,48.443,159.590
C04280=1024.599,361.121,357.316,171.976,48.444,159.591
C04281=1024.607,361.367,357.277,171.984,48.443,159.592
C04282=1024.614,361.614,357.238,171.991,48.444,159.594
C04283=1024.622,361.861,357.199,171.998,48.444,159.595
C04284=1024.630,362.108,357.160,172.007,48.444,159.596
C04285=1024.639,362.354,357.121,172.014,48.444,159.597
C04286=1024.646,362.601,357.083,172.022,48.444,159.598
C04287=1024.654,362.848,357.043,172.030,48.445,159.599
C04288=1024.662,363.095,357.004,172.037,48.445,159.600
C04289=1024.671,363.342,356.965,172.045,48.445,159.602
C04290=1024.679,363.588,356.926,172.052,48.445,159.603
C04291=1024.687,363.835,356.887,172.061,48.445,159.604
C04292=1024.695,364.082,356.847,172.068,48.446,159.605
C04293=1024.704,364.329,356.808,172.075,48.447,159.606
C04294=1024.711,364.575,356.769,172.083,48.446,159.608
C04295=1024.720,364.822,356.730,172.091,48.447,159.609
C04296=1024.728,365.069,356.691,172.099,48.447,159.610
C04297=1024.736,365.315,356.651,172.107,48.448,159.611
C04298=1024.744,365.548,356.614,172.114,48.448,159.612
C04299=1024.752,365.781,356.577,172.121,48.448,159.614
C04300=1024.760,366.014,356.540,172.129,48.448,159.615
C04301=1024.767,366.246,356.502,172.136,48.448,159.616
C04302=1024.776,366.479,356.465,172.144,48.449,159.617
C04303=1024.783,366.711,356.429,172.151,48.450,159.618
C04304=1024.791,366.944,356.391,172.158,48.450,159.619
C04305=1024.798,367.176,356.354,172.166,48.450,159.620
C04306=1024.807,367.423,356.315,172.174,48.450,159.622
C04307=1024.815,367.670,356.275,172.181,48.451,159.623
C04308=1024.824,367.917,356.236,172.190,48.451,159.624
C04309=1024.832,368.164,356.196,172.198,48.452,159.626
C04310=1024.841,368.410,356.156,172.206,48.452,159.627
C04311=1024.849,368.656,356.116,172.214,48.452,159.628
C04312=1024.857,368.903,356.076,172.222,48.454,159.629
C04313=1024.866,369.149,356.036,172.230,48.454,159.631
C04314=1024.874,369.397,355.996,172.238,48.454,159.632
C04315=1024.883,369.644,355.957,172.246,48.455,159.633
C04316=1024.891,369.890,355.916,172.254,48.456,159.635
C04317=1024.898,370.137,355.876,172.262,48.456,159.636
C04318=1024.907,370.383,355.836,172.271,48.456,159.637
C04319=1024.915,370.630,355.796,172.278,48.457,159.639
C04320=1024.924,370.876,355.756,172.287,48.458,159.640
C04321=1024.932,371.123,355.716,172.295,48.458,159.641
C04322=1024.941,371.369,355.676,172.303,48.459,159.643
C04323=1024.949,371.616,355.635,172.311,48.459,159.644
C04324=1024.958,371.863,355.595,172.320,48.460,159.645
C04325=1024.966,372.109,355.555,172.327,48.461,159.647
C04326=1024.974,372.356,355.514,172.336,48.462,159.648
C04327=1024.983,372.603,355.475,172.345,48.463,159.650
C04328=1024.991,372.849,355.434,172.352,48.463,159.651
C04329=1025.000,373.096,355.393,172.361,48.464,159.652
C04330=1025.008,373.342,355.353,172.369,48.464,159.654
C04331=1025.018,373.589,355.312,172.377,48.465,159.655
C04332=1025.026,373.835,355.272,172.386,48.466,159.656
C04333=1025.035,374.082,355.232,172.394,48.466,159.658
C04334=1025.043,374.328,355.191,172.403,48.467,159.659
C04335=1025.051,374.575,355.150,172.411,48.468,159.661
C04336=1025.060,374.821,355.110,172.419,48.469,159.662
C04337=1025.069,375.068,355.069,172.428,48.469,159.663
C04338=1025.078,375.314,355.029,172.437,48.470,159.665
C04339=1025.086,375.561,354.988,172.445,48.471,159.666
C04340=1025.095,375.807,354.948,172.453,48.472,159.668
C04341=1025.104,376.054,354.907,172.462,48.473,159.669
C04342=1025.113,376.300,354.866,172.471,48.474,159.671
C04343=1025.121,376.547,354.826,172.479,48.475,159.672
C04344=1025.130,376.794,354.785,172.488,48.476,159.674
C04345=1025.138,377.041,354.744,172.497,48.476,159.675
C04346=1025.148,377.286,354.703,172.504,48.478,159.677
C04347=1025.156,377.533,354.662,172.513,48.478,159.678
C04348=1025.165,377.779,354.620,172.522,48.479,159.680
C04349=1025.173,378.026,354.579,172.531,48.481,159.681
C04350=1025.182,378.272,354.538,172.540,48.482,159.683
C04351=1025.190,378.518,354.497,172.549,48.482,159.684
C04352=1025.199,378.765,354.455,172.557,48.483,159.686
C04353=1025.208,379.011,354.414,172.566,48.485,159.687
C04354=1025.217,379.258,354.373,172.575,48.485,159.689
C04355=1025.225,379.504,354.331,172.583,48.487,159.690
C04356=1025.235,379.750,354.290,172.592,48.488,159.692
C04357=1025.243,379.997,354.249,172.601,48.489,159.694
C04358=1025.252,380.239,354.208,172.609,48.490,159.695
C04359=1025.261,380.483,354.167,172.618,48.491,159.697
C04360=1025.269,380.727,354.126,172.627,48.492,159.698
C04361=1025.279,380.970,354.085,172.636,48.493,159.700
C04362=1025.287,381.213,354.044,172.645,48.494,159.701
C04363=1025.295,381.456,354.003,172.654,48.496,159.703
C04364=1025.305,381.699,353.962,172.663,48.496,159.705
C04365=1025.313,381.943,353.921,172.672,48.498,159.706
C04366=1025.322,382.190,353.879,172.681,48.499,159.708
C04367=1025.331,382.435,353.838,172.690,48.500,159.709
C04368=1025.340,382.682,353.796,172.699,48.501,159.711
C04369=1025.349,382.928,353.754,172.708,48.502,159.713
C04370=1025.358,383.174,353.713,172.717,48.504,159.714
C04371=1025.367,383.421,353.671,172.726,48.505,159.716
C04372=1025.376,383.667,353.628,172.735,48.506,159.718
C04373=1025.385,383.914,353.586,172.744,48.508,159.719
C04374=1025.395,384.160,353.545,172.754,48.508,159.721
C04375=1025.404,384.406,353.504,172.763,48.510,159.723
C04376=1025.413,384.652,353.461,172.772,48.511,159.724
C04377=1025.422,384.898,353.419,172.781,48.512,159.726
C04378=1025.431,385.144,353.378,172.790,48.514,159.728
C04379=1025.440,385.390,353.335,172.800,48.515,159.729
C04380=1025.450,385.637,353.293,172.809,48.516,159.731
C04381=1025.459,385.884,353.252,172.818,48.518,159.733
C04382=1025.468,386.129,353.209,172.827,48.519,159.735
C04383=1025.477,386.375,353.167,172.837,48.520,159.736
C04384=1025.487,386.622,353.125,172.847,48.522,159.738
C04385=1025.496,386.868,353.082,172.856,48.524,159.740
C04386=1025.505,387.114,353.040,172.865,48.525,159.742
C04387=1025.513,387.360,352.997,172.874,48.526,159.743
C04388=1025.523,387.607,352.955,172.885,48.528,159.745
C04389=1025.532,387.852,352.912,172.894,48.529,159.747
C04390=1025.542,388.098,352.870,172.903,48.531,159.749
C04391=1025.552,388.345,352.827,172.913,48.532,159.751
C04392=1025.560,388.591,352.785,172.922,48.534,159.752
C04393=1025.569,388.837,352.742,172.932,48.536,159.754
C04394=1025.579,389.084,352.699,172.942,48.537,159.756
C04395=1025.588,389.329,352.657,172.951,48.539,159.758
C04396=1025.597,389.576,352.614,172.961,48.541,159.760
C04397=1025.607,389.821,352.570,172.971,48.542,159.761
C04398=1025.617,390.068,352.528,172.980,48.544,159.763
C04399=1025.625,390.314,352.485,172.989,48.545,159.765
C04400=1025.635,390.560,352.442,173.000,48.547,159.767
C04401=1025.644,390.806,352.399,173.009,48.549,159.769
C04402=1025.654,391.052,352.355,173.020,48.550,159.771
C04403=1025.663,391.298,352.313,173.029,48.552,159.773
C04404=1025.673,391.544,352.270,173.039,48.553,159.775
C04405=1025.681,391.790,352.226,173.049,48.555,159.776
C04406=1025.691,392.036,352.184,173.059,48.557,159.778
C04407=1025.701,392.282,352.141,173.069,48.559,159.780
C04408=1025.710,392.528,352.097,173.079,48.560,159.782
C04409=1025.720,392.774,352.054,173.089,48.562,159.784
C04410=1025.729,393.019,352.011,173.099,48.564,159.786
C04411=1025.739,393.266,351.967,173.108,48.566,159.788
C04412=1025.749,393.512,351.924,173.119,48.567,159.790
C04413=1025.758,393.758,351.880,173.128,48.569,159.792
C04414=1025.768,394.003,351.837,173.139,48.572,159.794
C04415=1025.777,394.250,351.793,173.150,48.573,159.796
C04416=1025.787,394.496,351.750,173.159,48.575,159.798
C04417=1025.796,394.742,351.706,173.170,48.577,159.800
C04418=1025.810,395.091,351.644,173.184,48.580,159.803
C04419=1025.824,395.440,351.582,173.199,48.582,159.806
C04420=1025.837,395.789,351.520,173.213,48.586,159.809
C04421=1025.851,396.139,351.458,173.227,48.588,159.811
C04422=1025.861,396.385,351.414,173.238,48.590,159.814
C04423=1025.871,396.631,351.370,173.248,48.592,159.815
C04424=1025.880,396.877,351.326,173.259,48.594,159.818
C04425=1025.891,397.122,351.282,173.269,48.596,159.820
C04426=1025.900,397.368,351.238,173.280,48.598,159.822
C04427=1025.910,397.614,351.194,173.290,48.600,159.824
C04428=1025.919,397.860,351.150,173.301,48.602,159.826
C04429=1025.930,398.105,351.106,173.311,48.604,159.828
C04430=1025.939,398.351,351.062,173.321,48.606,159.830
C04431=1025.949,398.597,351.017,173.332,48.609,159.832
C04432=1025.959,398.843,350.973,173.343,48.611,159.834
C04433=1025.969,399.089,350.929,173.354,48.613,159.837
C04434=1025.978,399.334,350.884,173.365,48.615,159.839
C04435=1025.989,399.580,350.840,173.375,48.617,159.841
C04436=1025.999,399.826,350.796,173.385,48.620,159.843
C04437=1026.009,400.072,350.751,173.396,48.622,159.845
C04438=1026.018,400.318,350.706,173.407,48.624,159.847
C04439=1026.029,400.563,350.662,173.418,48.626,159.850
C04440=1026.039,400.810,350.617,173.428,48.628,159.852
C04441=1026.048,401.055,350.573,173.439,48.630,159.854
C04442=1026.057,401.264,350.534,173.449,48.632,159.856
C04443=1026.065,401.474,350.496,173.458,48.634,159.858
C04444=1026.074,401.683,350.458,173.468,48.636,159.860
C04445=1026.083,401.893,350.420,173.476,48.639,159.862
C04446=1026.091,402.102,350.381,173.486,48.641,159.864
C04447=1026.100,402.312,350.344,173.495,48.643,159.866
C04448=1026.108,402.521,350.305,173.505,48.644,159.867
C04449=1026.117,402.731,350.266,173.514,48.646,159.869
C04450=1026.126,402.976,350.221,173.525,48.649,159.872
C04451=1026.137,403.222,350.176,173.536,48.651,159.874
C04452=1026.146,403.468,350.131,173.547,48.654,159.876
C04453=1026.156,403.713,350.085,173.559,48.657,159.879
C04454=1026.167,403.959,350.040,173.569,48.659,159.881
C04455=1026.177,404.204,349.996,173.581,48.661,159.883
C04456=1026.188,404.450,349.950,173.593,48.664,159.886
C04457=1026.198,404.696,349.905,173.604,48.666,159.888
C04458=1026.208,404.941,349.859,173.615,48.669,159.890
C04459=1026.219,405.187,349.814,173.626,48.671,159.893
C04460=1026.229,405.432,349.769,173.637,48.674,159.895
C04461=1026.239,405.678,349.723,173.649,48.676,159.898
C04462=1026.250,405.924,349.678,173.660,48.679,159.900
C04463=1026.260,406.169,349.632,173.671,48.682,159.902
C04464=1026.270,406.415,349.587,173.684,48.684,159.905
C04465=1026.280,406.661,349.541,173.695,48.687,159.907
C04466=1026.291,406.906,349.495,173.706,48.689,159.910
C04467=1026.301,407.151,349.449,173.718,48.692,159.912
C04468=1026.312,407.397,349.404,173.730,48.695,159.915
C04469=1026.322,407.642,349.358,173.741,48.698,159.917
C04470=1026.333,407.888,349.312,173.753,48.700,159.919
C04471=1026.343,408.134,349.267,173.764,48.703,159.922
C04472=1026.354,408.380,349.221,173.777,48.706,159.925
C04473=1026.365,408.625,349.175,173.788,48.708,159.927
C04474=1026.375,408.870,349.128,173.800,48.711,159.929
C04475=1026.386,409.116,349.082,173.812,48.714,159.932
C04476=1026.397,409.361,349.036,173.824,48.716,159.934
C04477=1026.407,409.607,348.990,173.835,48.719,159.937
C04478=1026.421,409.905,348.934,173.851,48.723,159.940
C04479=1026.433,410.205,348.879,173.865,48.726,159.943
C04480=1026.446,410.504,348.821,173.879,48.730,159.946
C04481=1026.460,410.803,348.765,173.894,48.733,159.950
C04482=1026.470,411.048,348.718,173.905,48.736,159.952
C04483=1026.480,411.294,348.672,173.918,48.739,159.955
C04484=1026.491,411.539,348.625,173.930,48.742,159.958
C04485=1026.503,411.784,348.578,173.942,48.745,159.960
C04486=1026.513,412.030,348.532,173.955,48.748,159.963
C04487=1026.524,412.275,348.485,173.967,48.751,159.965
C04488=1026.535,412.520,348.439,173.980,48.754,159.968
C04489=1026.545,412.766,348.391,173.991,48.757,159.971
C04490=1026.556,413.011,348.344,174.004,48.760,159.974
C04491=1026.567,413.256,348.298,174.017,48.763,159.976
C04492=1026.579,413.502,348.251,174.029,48.766,159.979
C04493=1026.589,413.747,348.204,174.042,48.769,159.982
C04494=1026.600,413.993,348.157,174.054,48.773,159.984
C04495=1026.611,414.238,348.110,174.066,48.776,159.987
C04496=1026.622,414.483,348.063,174.079,48.779,159.990
C04497=1026.633,414.729,348.016,174.092,48.782,159.993
C04498=1026.645,414.974,347.969,174.104,48.785,159.996
C04499=1026.655,415.220,347.922,174.117,48.788,159.998
C04500=1026.667,415.465,347.874,174.130,48.791,160.001
C04501=1026.678,415.710,347.827,174.142,48.794,160.004
C04502=1026.689,415.955,347.780,174.155,48.798,160.007
C04503=1026.700,416.201,347.732,174.168,48.801,160.010
C04504=1026.712,416.445,347.685,174.181,48.804,160.013
C04505=1026.722,416.691,347.637,174.194,48.808,160.015
C04506=1026.733,416.936,347.589,174.207,48.811,160.018
C04507=1026.745,417.181,347.541,174.220,48.815,160.021
C04508=1026.755,417.427,347.494,174.233,48.818,160.024
C04509=1026.767,417.672,347.446,174.246,48.821,160.027
C04510=1026.778,417.916,347.398,174.260,48.824,160.030
C04511=1026.790,418.161,347.350,174.272,48.828,160.033
C04512=1026.801,418.407,347.302,174.285,48.831,160.036
C04513=1026.812,418.652,347.254,174.299,48.835,160.039
C04514=1026.824,418.897,347.206,174.312,48.838,160.042
C04515=1026.835,419.143,347.158,174.325,48.841,160.045
C04516=1026.847,419.388,347.110,174.339,48.845,160.048
C04517=1026.858,419.633,347.062,174.352,48.849,160.051
C04518=1026.869,419.878,347.014,174.366,48.852,160.054
C04519=1026.881,420.123,346.965,174.379,48.855,160.057
C04520=1026.893,420.368,346.917,174.392,48.859,160.060
C04521=1026.904,420.613,346.869,174.406,48.862,160.063
C04522=1026.915,420.858,346.820,174.419,48.866,160.066
C04523=1026.927,421.103,346.772,174.434,48.870,160.069
C04524=1026.938,421.348,346.724,174.447,48.874,160.072
C04525=1026.950,421.593,346.676,174.461,48.877,160.075
C04526=1026.962,421.839,346.627,174.474,48.881,160.078
C04527=1026.974,422.083,346.579,174.488,48.884,160.081
C04528=1026.986,422.328,346.530,174.502,48.888,160.085
C04529=1026.997,422.573,346.481,174.516,48.891,160.088
C04530=1027.009,422.819,346.432,174.530,48.895,160.091
C04531=1027.021,423.063,346.384,174.544,48.899,160.094
C04532=1027.032,423.308,346.334,174.558,48.903,160.097
C04533=1027.044,423.553,346.285,174.572,48.906,160.101
C04534=1027.056,423.798,346.236,174.586,48.911,160.104
C04535=1027.067,424.043,346.187,174.600,48.914,160.107
C04536=1027.080,424.288,346.138,174.615,48.918,160.110
C04537=1027.091,424.533,346.089,174.629,48.922,160.114
C04538=1027.106,424.842,346.027,174.647,48.927,160.118
C04539=1027.122,425.152,345.965,174.665,48.932,160.122
C04540=1027.137,425.462,345.902,174.683,48.937,160.126
C04541=1027.151,425.771,345.840,174.701,48.942,160.130
C04542=1027.164,426.016,345.790,174.716,48.946,160.134
C04543=1027.176,426.261,345.741,174.730,48.949,160.137
C04544=1027.188,426.505,345.691,174.745,48.953,160.140
C04545=1027.200,426.750,345.641,174.759,48.957,160.144
C04546=1027.212,426.996,345.592,174.774,48.962,160.147
C04547=1027.224,427.240,345.542,174.789,48.966,160.151
C04548=1027.236,427.484,345.492,174.804,48.970,160.154
C04549=1027.249,427.729,345.442,174.819,48.974,160.158
C04550=1027.261,427.974,345.392,174.834,48.978,160.161
C04551=1027.273,428.218,345.342,174.849,48.982,160.165
C04552=1027.285,428.463,345.292,174.864,48.986,160.168
C04553=1027.297,428.708,345.242,174.879,48.991,160.172
C04554=1027.309,428.953,345.191,174.893,48.995,160.175
C04555=1027.321,429.198,345.141,174.909,48.999,160.179
C04556=1027.334,429.442,345.090,174.924,49.003,160.182
C04557=1027.346,429.687,345.040,174.939,49.007,160.186
C04558=1027.359,429.932,344.990,174.955,49.012,160.190
C04559=1027.371,430.176,344.939,174.970,49.016,160.193
C04560=1027.384,430.421,344.889,174.986,49.020,160.197
C04561=1027.396,430.665,344.838,175.001,49.024,160.200
C04562=1027.408,430.910,344.788,175.016,49.029,160.204
C04563=1027.422,431.155,344.737,175.032,49.033,160.208
C04564=1027.434,431.399,344.686,175.047,49.037,160.211
C04565=1027.447,431.644,344.636,175.063,49.042,160.215
C04566=1027.459,431.888,344.585,175.079,49.046,160.219
C04567=1027.472,432.133,344.534,175.095,49.051,160.222
C04568=1027.485,432.377,344.483,175.111,49.055,160.226
C04569=1027.498,432.621,344.432,175.127,49.059,160.230
C04570=1027.511,432.866,344.381,175.142,49.064,160.234
C04571=1027.524,433.110,344.330,175.158,49.068,160.237
C04572=1027.537,433.355,344.279,175.174,49.073,160.241
C04573=1027.549,433.599,344.228,175.191,49.077,160.245
C04574=1027.563,433.844,344.177,175.206,49.082,160.249
C04575=1027.576,434.088,344.126,175.222,49.086,160.253
C04576=1027.588,434.333,344.074,175.239,49.091,160.257
C04577=1027.601,434.577,344.023,175.255,49.096,160.261
C04578=1027.614,434.822,343.971,175.272,49.100,160.264
C04579=1027.627,435.066,343.920,175.288,49.105,160.268
C04580=1027.640,435.310,343.869,175.304,49.110,160.272
C04581=1027.653,435.555,343.816,175.321,49.114,160.276
C04582=1027.666,435.799,343.765,175.337,49.119,160.280
C04583=1027.679,436.043,343.713,175.354,49.124,160.284
C04584=1027.692,436.288,343.661,175.370,49.129,160.288
C04585=1027.706,436.532,343.609,175.388,49.133,160.292
C04586=1027.718,436.776,343.557,175.405,49.138,160.296
C04587=1027.732,437.020,343.506,175.421,49.142,160.300
C04588=1027.745,437.264,343.453,175.438,49.148,160.304
C04589=1027.758,437.509,343.401,175.456,49.152,160.309
C04590=1027.772,437.752,343.349,175.472,49.157,160.312
C04591=1027.785,437.997,343.296,175.489,49.162,160.317
C04592=1027.798,438.241,343.244,175.507,49.167,160.321
C04593=1027.812,438.485,343.192,175.524,49.172,160.325
C04594=1027.825,438.729,343.139,175.541,49.177,160.329
C04595=1027.839,438.973,343.086,175.558,49.182,160.333
C04596=1027.852,439.217,343.035,175.576,49.186,160.337
C04597=1027.866,439.461,342.981,175.593,49.192,160.342
C04598=1027.879,439.709,342.928,175.611,49.197,160.346
C04599=1027.893,439.957,342.874,175.629,49.202,160.350
C04600=1027.907,440.205,342.821,175.647,49.207,160.355
C04601=1027.921,440.452,342.767,175.664,49.212,160.359
C04602=1027.935,440.697,342.713,175.682,49.217,160.363
C04603=1027.949,440.940,342.661,175.700,49.223,160.368
C04604=1027.962,441.184,342.608,175.718,49.227,160.372
C04605=1027.976,441.429,342.555,175.736,49.232,160.377
C04606=1027.990,441.672,342.502,175.755,49.238,160.381
C04607=1028.004,441.917,342.448,175.773,49.243,160.385
C04608=1028.018,442.160,342.395,175.791,49.248,160.390
C04609=1028.032,442.405,342.342,175.809,49.253,160.394
C04610=1028.045,442.647,342.289,175.827,49.258,160.399
C04611=1028.060,442.890,342.236,175.846,49.263,160.403
C04612=1028.075,443.134,342.183,175.864,49.269,160.408
C04613=1028.089,443.377,342.130,175.882,49.274,160.412
C04614=1028.105,443.620,342.078,175.900,49.279,160.416
C04615=1028.121,443.863,342.027,175.919,49.284,160.421
C04616=1028.138,444.108,341.975,175.938,49.288,160.425
C04617=1028.154,444.352,341.925,175.957,49.293,160.430
C04618=1028.172,444.595,341.874,175.976,49.298,160.434
C04619=1028.189,444.839,341.824,175.995,49.303,160.439
C04620=1028.208,445.083,341.774,176.014,49.308,160.443
C04621=1028.227,445.327,341.725,176.033,49.312,160.448
C04622=1028.246,445.571,341.676,176.052,49.316,160.452
C04623=1028.266,445.815,341.629,176.072,49.321,160.457
C04624=1028.286,446.059,341.580,176.091,49.325,160.461
C04625=1028.306,446.303,341.532,176.111,49.329,160.465
C04626=1028.327,446.548,341.485,176.130,49.333,160.470
C04627=1028.349,446.792,341.438,176.150,49.338,160.474
C04628=1028.371,447.037,341.392,176.170,49.341,160.478
C04629=1028.393,447.282,341.346,176.190,49.345,160.483
C04630=1028.417,447.526,341.300,176.210,49.349,160.487
C04631=1028.440,447.771,341.255,176.229,49.353,160.491
C04632=1028.464,448.016,341.210,176.249,49.357,160.496
C04633=1028.488,448.261,341.166,176.270,49.360,160.500
C04634=1028.513,448.505,341.121,176.290,49.364,160.505
C04635=1028.539,448.751,341.078,176.310,49.367,160.509
C04636=1028.565,448.996,341.034,176.331,49.371,160.513
C04637=1028.591,449.240,340.992,176.351,49.375,160.518
C04638=1028.618,449.486,340.949,176.372,49.378,160.522
C04639=1028.645,449.731,340.908,176.393,49.381,160.526
C04640=1028.672,449.976,340.866,176.413,49.385,160.531
C04641=1028.701,450.222,340.825,176.435,49.387,160.535
C04642=1028.729,450.467,340.783,176.456,49.391,160.539
C04643=1028.759,450.713,340.743,176.476,49.394,160.544
C04644=1028.788,450.958,340.703,176.498,49.397,160.548
C04645=1028.818,451.203,340.663,176.519,49.399,160.552
C04646=1028.848,451.448,340.624,176.540,49.403,160.557
C04647=1028.880,451.694,340.585,176.562,49.405,160.561
C04648=1028.911,451.940,340.547,176.583,49.408,160.565
C04649=1028.943,452.185,340.509,176.605,49.410,160.569
C04650=1028.976,452.431,340.471,176.626,49.413,160.574
C04651=1029.008,452.677,340.434,176.649,49.416,160.578
C04652=1029.042,452.922,340.397,176.670,49.418,160.582
C04653=1029.075,453.168,340.361,176.692,49.421,160.587
C04654=1029.110,453.414,340.325,176.715,49.423,160.591
C04655=1029.145,453.660,340.289,176.737,49.425,160.595
C04656=1029.180,453.905,340.254,176.759,49.428,160.600
C04657=1029.216,454.151,340.219,176.781,49.430,160.604
C04658=1028.939,454.225,339.883,176.784,49.492,160.624
C04659=1028.903,453.979,339.918,176.762,49.489,160.620
C04660=1028.868,453.733,339.953,176.739,49.487,160.615
C04661=1028.833,453.488,339.989,176.717,49.485,160.611
C04662=1028.798,453.241,340.025,176.695,49.483,160.607
C04663=1028.765,452.996,340.061,176.673,49.480,160.602
C04664=1028.731,452.751,340.098,176.651,49.478,160.598
C04665=1028.697,452.505,340.134,176.629,49.476,160.594
C04666=1028.665,452.259,340.172,176.607,49.473,160.589
C04667=1028.633,452.014,340.210,176.586,49.470,160.585
C04668=1028.601,451.769,340.248,176.564,49.467,160.581
C04669=1028.570,451.523,340.287,176.543,49.465,160.577
C04670=1028.539,451.277,340.326,176.521,49.462,160.572
C04671=1028.510,451.032,340.366,176.499,49.460,160.568
C04672=1028.480,450.786,340.405,176.479,49.456,160.564
C04673=1028.451,450.540,340.446,176.457,49.454,160.559
C04674=1028.422,450.295,340.486,176.436,49.450,160.555
C04675=1028.393,450.049,340.527,176.415,49.448,160.551
C04676=1028.365,449.805,340.569,176.394,49.444,160.546
C04677=1028.339,449.559,340.611,176.373,49.441,160.542
C04678=1028.310,449.314,340.653,176.353,49.438,160.538
C04679=1028.284,449.069,340.696,176.332,49.435,160.533
C04680=1028.258,448.824,340.739,176.311,49.431,160.529
C04681=1028.233,448.579,340.782,176.291,49.428,160.525
C04682=1028.208,448.334,340.825,176.271,49.425,160.520
C04683=1028.183,448.089,340.871,176.250,49.421,160.516
C04684=1028.159,447.844,340.915,176.230,49.418,160.512
C04685=1028.136,447.599,340.961,176.210,49.413,160.507
C04686=1028.113,447.355,341.006,176.190,49.410,160.503
C04687=1028.090,447.110,341.052,176.171,49.406,160.499
C04688=1028.068,446.866,341.098,176.151,49.402,160.494
C04689=1028.046,446.621,341.145,176.131,49.398,160.490
C04690=1028.025,446.377,341.191,176.111,49.394,160.485
C04691=1028.004,446.133,341.239,176.091,49.391,160.481
C04692=1027.983,445.888,341.287,176.072,49.386,160.477
C04693=1027.964,445.644,341.335,176.052,49.382,160.472
C04694=1027.944,445.400,341.383,176.033,49.378,160.468
C04695=1027.925,445.155,341.433,176.014,49.373,160.463
C04696=1027.906,444.911,341.482,175.995,49.369,160.459
C04697=1027.889,444.668,341.532,175.976,49.364,160.455
C04698=1027.870,444.424,341.582,175.957,49.360,160.450
C04699=1027.854,444.180,341.633,175.938,49.355,160.446
C04700=1027.837,443.937,341.684,175.919,49.350,160.441
C04701=1027.820,443.693,341.735,175.901,49.345,160.437
C04702=1027.804,443.450,341.787,175.881,49.341,160.432
C04703=1027.790,443.206,341.839,175.863,49.336,160.428
C04704=1027.774,442.963,341.892,175.844,49.331,160.423
C04705=1027.760,442.719,341.945,175.826,49.326,160.419
C04706=1027.746,442.476,341.998,175.808,49.321,160.415
C04707=1027.732,442.233,342.051,175.790,49.316,160.410
C04708=1027.718,441.988,342.105,175.772,49.311,160.406
C04709=1027.705,441.745,342.157,175.753,49.306,160.401
C04710=1027.691,441.502,342.211,175.735,49.300,160.397
C04711=1027.677,441.260,342.264,175.717,49.295,160.392
C04712=1027.663,441.019,342.316,175.699,49.291,160.388
C04713=1027.649,440.778,342.368,175.682,49.286,160.384
C04714=1027.636,440.536,342.421,175.664,49.280,160.380
C04715=1027.623,440.295,342.473,175.646,49.276,160.375
C04716=1027.609,440.053,342.525,175.629,49.271,160.371
C04717=1027.595,439.812,342.577,175.612,49.266,160.367
C04718=1027.582,439.570,342.630,175.595,49.261,160.363
C04719=1027.569,439.327,342.682,175.577,49.256,160.359
C04720=1027.555,439.083,342.735,175.559,49.251,160.354
C04721=1027.542,438.839,342.787,175.542,49.246,160.350
C04722=1027.528,438.595,342.840,175.524,49.241,160.346
C04723=1027.515,438.350,342.892,175.508,49.237,160.342
C04724=1027.501,438.106,342.945,175.490,49.232,160.338
C04725=1027.487,437.862,342.997,175.473,49.227,160.333
C04726=1027.475,437.617,343.050,175.455,49.222,160.329
C04727=1027.461,437.373,343.102,175.439,49.218,160.325
C04728=1027.448,437.129,343.153,175.422,49.213,160.321
C04729=1027.434,436.886,343.206,175.404,49.208,160.317
C04730=1027.421,436.641,343.258,175.388,49.203,160.313
C04731=1027.408,436.397,343.310,175.371,49.199,160.309
C04732=1027.395,436.152,343.361,175.355,49.194,160.305
C04733=1027.383,435.908,343.414,175.337,49.190,160.301
C04734=1027.369,435.664,343.465,175.320,49.185,160.297
C04735=1027.355,435.419,343.517,175.304,49.180,160.293
C04736=1027.343,435.175,343.568,175.288,49.176,160.289
C04737=1027.330,434.931,343.621,175.271,49.171,160.285
C04738=1027.317,434.686,343.672,175.255,49.166,160.281
C04739=1027.304,434.442,343.723,175.239,49.162,160.278
C04740=1027.291,434.197,343.774,175.222,49.158,160.274
C04741=1027.278,433.954,343.826,175.206,49.153,160.270
C04742=1027.265,433.708,343.878,175.190,49.149,160.266
C04743=1027.253,433.464,343.929,175.173,49.144,160.262
C04744=1027.239,433.220,343.980,175.158,49.139,160.258
C04745=1027.227,432.976,344.031,175.142,49.135,160.255
C04746=1027.213,432.731,344.082,175.126,49.131,160.251
C04747=1027.201,432.486,344.133,175.109,49.127,160.247
C04748=1027.188,432.242,344.183,175.094,49.122,160.243
C04749=1027.175,431.997,344.235,175.078,49.118,160.240
C04750=1027.163,431.753,344.285,175.062,49.114,160.236
C04751=1027.150,431.508,344.336,175.047,49.109,160.232
C04752=1027.137,431.263,344.387,175.031,49.105,160.229
C04753=1027.124,431.019,344.437,175.015,49.101,160.225
C04754=1027.112,430.775,344.488,175.000,49.097,160.221
C04755=1027.099,430.530,344.538,174.984,49.093,160.217
C04756=1027.087,430.286,344.589,174.969,49.088,160.214
C04757=1027.075,430.041,344.639,174.953,49.084,160.210
C04758=1027.062,429.797,344.690,174.938,49.080,160.207
C04759=1027.050,429.552,344.740,174.922,49.076,160.203
C04760=1027.037,429.307,344.790,174.907,49.072,160.200
C04761=1027.025,429.062,344.840,174.892,49.068,160.196
C04762=1027.012,428.818,344.891,174.876,49.064,160.192
C04763=1027.000,428.573,344.941,174.862,49.060,160.189
C04764=1026.988,428.328,344.991,174.847,49.055,160.185
C04765=1026.975,428.083,345.041,174.832,49.051,160.182
C04766=1026.964,427.839,345.091,174.816,49.048,160.179
C04767=1026.951,427.594,345.141,174.802,49.044,160.175
C04768=1026.939,427.350,345.191,174.787,49.040,160.172
C04769=1026.927,427.104,345.241,174.772,49.036,160.168
C04770=1026.915,426.860,345.290,174.758,49.032,160.165
C04771=1026.903,426.615,345.341,174.743,49.028,160.161
C04772=1026.891,426.370,345.391,174.728,49.024,160.158
C04773=1026.879,426.126,345.440,174.714,49.020,160.155
C04774=1026.867,425.881,345.490,174.699,49.016,160.151
C04775=1026.851,425.569,345.552,174.680,49.011,160.147
C04776=1026.836,425.257,345.616,174.661,49.006,160.143
C04777=1026.820,424.945,345.678,174.644,49.001,160.139
C04778=1026.806,424.633,345.741,174.625,48.996,160.134
C04779=1026.794,424.389,345.790,174.611,48.993,160.131
C04780=1026.781,424.143,345.839,174.597,48.988,160.128
C04781=1026.770,423.899,345.888,174.583,48.985,160.125
C04782=1026.758,423.653,345.937,174.568,48.981,160.121
C04783=1026.747,423.408,345.986,174.554,48.978,160.118
C04784=1026.735,423.164,346.035,174.540,48.974,160.115
C04785=1026.722,422.919,346.084,174.526,48.970,160.112
C04786=1026.711,422.674,346.133,174.512,48.967,160.108
C04787=1026.700,422.429,346.182,174.497,48.963,160.105
C04788=1026.688,422.184,346.231,174.484,48.959,160.102
C04789=1026.676,421.939,346.279,174.470,48.956,160.099
C04790=1026.665,421.693,346.328,174.457,48.952,160.096
C04791=1026.652,421.449,346.376,174.443,48.949,160.093
C04792=1026.641,421.203,346.424,174.428,48.945,160.090
C04793=1026.629,420.959,346.473,174.415,48.942,160.087
C04794=1026.618,420.713,346.521,174.401,48.938,160.084
C04795=1026.606,420.468,346.570,174.388,48.935,160.080
C04796=1026.594,420.223,346.618,174.375,48.931,160.078
C04797=1026.583,419.978,346.666,174.361,48.928,160.074
C04798=1026.571,419.733,346.714,174.348,48.924,160.071
C04799=1026.560,419.487,346.762,174.334,48.921,160.068
C04800=1026.548,419.242,346.810,174.320,48.917,160.065
C04801=1026.537,418.998,346.859,174.307,48.914,160.062
C04802=1026.526,418.753,346.906,174.294,48.911,160.059
C04803=1026.515,418.508,346.955,174.281,48.908,160.057
C04804=1026.504,418.263,347.003,174.267,48.904,160.053
C04805=1026.492,418.017,347.050,174.253,48.901,160.050
C04806=1026.481,417.771,347.098,174.241,48.897,160.048
C04807=1026.470,417.527,347.146,174.228,48.894,160.045
C04808=1026.459,417.282,347.194,174.215,48.891,160.042
C04809=1026.447,417.037,347.242,174.202,48.887,160.039
C04810=1026.436,416.791,347.289,174.189,48.885,160.036
C04811=1026.425,416.546,347.337,174.175,48.882,160.033
C04812=1026.414,416.301,347.385,174.162,48.878,160.030
C04813=1026.403,416.056,347.432,174.149,48.875,160.027
C04814=1026.392,415.811,347.480,174.137,48.872,160.025
C04815=1026.380,415.565,347.527,174.124,48.869,160.022
C04816=1026.369,415.320,347.573,174.111,48.865,160.019
C04817=1026.358,415.074,347.621,174.098,48.862,160.016
C04818=1026.347,414.829,347.669,174.086,48.859,160.013
C04819=1026.336,414.584,347.715,174.073,48.856,160.011
C04820=1026.325,414.339,347.763,174.060,48.853,160.008
C04821=1026.314,414.093,347.810,174.048,48.850,160.005
C04822=1026.303,413.848,347.856,174.035,48.847,160.002
C04823=1026.291,413.602,347.903,174.022,48.844,160.000
C04824=1026.281,413.357,347.950,174.011,48.841,159.997
C04825=1026.270,413.111,347.997,173.998,48.838,159.994
C04826=1026.259,412.866,348.044,173.985,48.835,159.991
C04827=1026.249,412.621,348.091,173.973,48.832,159.989
C04828=1026.238,412.376,348.138,173.960,48.829,159.986
C04829=1026.226,412.131,348.185,173.948,48.826,159.983
C04830=1026.215,411.885,348.231,173.936,48.823,159.981
C04831=1026.205,411.640,348.278,173.924,48.820,159.978
C04832=1026.194,411.395,348.325,173.911,48.818,159.976
C04833=1026.183,411.148,348.371,173.900,48.815,159.973
C04834=1026.172,410.903,348.417,173.887,48.812,159.970
C04835=1026.160,410.602,348.475,173.872,48.809,159.967
C04836=1026.147,410.301,348.531,173.858,48.805,159.964
C04837=1026.134,410.000,348.589,173.843,48.802,159.961
C04838=1026.121,409.699,348.646,173.829,48.798,159.958
C04839=1026.110,409.453,348.691,173.816,48.796,159.955
C04840=1026.099,409.207,348.738,173.804,48.793,159.953
C04841=1026.088,408.961,348.784,173.792,48.790,159.950
C04842=1026.078,408.716,348.830,173.780,48.788,159.948
C04843=1026.068,408.471,348.875,173.769,48.785,159.945
C04844=1026.057,408.225,348.921,173.756,48.782,159.942
C04845=1026.046,407.979,348.967,173.745,48.779,159.940
C04846=1026.036,407.734,349.013,173.733,48.777,159.938
C04847=1026.025,407.488,349.059,173.722,48.775,159.935
C04848=1026.014,407.243,349.105,173.710,48.772,159.933
C04849=1026.004,406.997,349.150,173.699,48.770,159.930
C04850=1025.992,406.752,349.196,173.687,48.767,159.928
C04851=1025.983,406.506,349.241,173.675,48.765,159.925
C04852=1025.972,406.261,349.287,173.664,48.762,159.923
C04853=1025.962,406.015,349.332,173.652,48.760,159.921
C04854=1025.952,405.770,349.377,173.641,48.757,159.918
C04855=1025.941,405.524,349.423,173.629,48.754,159.916
C04856=1025.931,405.278,349.469,173.617,48.752,159.913
C04857=1025.921,405.033,349.514,173.606,48.750,159.911
C04858=1025.910,404.787,349.560,173.595,48.747,159.909
C04859=1025.900,404.541,349.605,173.584,48.744,159.906
C04860=1025.890,404.296,349.650,173.572,48.742,159.904
C04861=1025.880,404.050,349.696,173.561,48.740,159.902
C04862=1025.870,403.804,349.741,173.550,48.737,159.899
C04863=1025.859,403.559,349.786,173.539,48.735,159.897
C04864=1025.850,403.313,349.831,173.528,48.732,159.895
C04865=1025.840,403.068,349.876,173.517,48.730,159.892
C04866=1025.829,402.822,349.921,173.505,48.728,159.890
C04867=1025.819,402.576,349.966,173.494,48.726,159.888
C04868=1025.808,402.331,350.011,173.483,48.723,159.885
C04869=1025.799,402.085,350.056,173.472,48.721,159.883
C04870=1025.789,401.840,350.101,173.461,48.719,159.881
C04871=1025.779,401.594,350.146,173.450,48.717,159.879
C04872=1025.769,401.348,350.191,173.439,48.714,159.876
C04873=1025.759,401.103,350.236,173.428,48.712,159.874
C04874=1025.750,400.856,350.280,173.418,48.710,159.872
C04875=1025.739,400.611,350.325,173.407,48.708,159.870
C04876=1025.729,400.365,350.369,173.396,48.705,159.868
C04877=1025.719,400.120,350.414,173.385,48.703,159.866
C04878=1025.710,399.873,350.458,173.374,48.701,159.863
C04879=1025.699,399.628,350.503,173.363,48.699,159.861
C04880=1025.689,399.382,350.548,173.353,48.697,159.859
C04881=1025.680,399.136,350.592,173.342,48.695,159.857
C04882=1025.669,398.891,350.636,173.331,48.693,159.855
C04883=1025.660,398.644,350.680,173.321,48.691,159.853
C04884=1025.650,398.399,350.725,173.310,48.689,159.850
C04885=1025.640,398.153,350.769,173.300,48.686,159.848
C04886=1025.631,397.907,350.813,173.289,48.685,159.846
C04887=1025.620,397.662,350.857,173.279,48.683,159.844
C04888=1025.611,397.416,350.901,173.268,48.681,159.842
C04889=1025.601,397.170,350.945,173.257,48.679,159.840
C04890=1025.591,396.924,350.989,173.247,48.677,159.838
C04891=1025.581,396.678,351.033,173.237,48.675,159.836
C04892=1025.571,396.432,351.077,173.226,48.673,159.834
C04893=1025.562,396.186,351.121,173.216,48.671,159.832
C04894=1025.552,395.940,351.165,173.205,48.670,159.830
C04895=1025.541,395.662,351.215,173.193,48.667,159.827
C04896=1025.530,395.382,351.264,173.182,48.665,159.825
C04897=1025.519,395.103,351.313,173.171,48.663,159.823
C04898=1025.508,394.825,351.363,173.158,48.661,159.820
C04899=1025.499,394.578,351.407,173.149,48.659,159.819
C04900=1025.489,394.333,351.450,173.138,48.657,159.817
C04901=1025.480,394.086,351.494,173.128,48.655,159.815
C04902=1025.470,393.841,351.537,173.119,48.654,159.813
C04903=1025.461,393.595,351.581,173.108,48.652,159.811
C04904=1025.451,393.348,351.624,173.098,48.650,159.809
C04905=1025.441,393.102,351.668,173.088,48.648,159.807
C04906=1025.432,392.857,351.711,173.078,48.647,159.805
C04907=1025.422,392.610,351.754,173.068,48.645,159.803
C04908=1025.413,392.364,351.798,173.058,48.643,159.801
C04909=1025.403,392.119,351.840,173.047,48.642,159.799
C04910=1025.393,391.872,351.883,173.038,48.640,159.797
C04911=1025.385,391.627,351.927,173.027,48.638,159.795
C04912=1025.375,391.380,351.970,173.018,48.637,159.793
C04913=1025.365,391.134,352.013,173.008,48.635,159.791
C04914=1025.356,390.888,352.056,172.998,48.633,159.790
C04915=1025.341,390.506,352.123,172.983,48.631,159.787
C04916=1025.327,390.123,352.189,172.968,48.629,159.784
C04917=1025.313,389.741,352.256,172.952,48.626,159.781
C04918=1025.298,389.359,352.323,172.937,48.624,159.778
C04919=1025.289,389.113,352.366,172.928,48.622,159.776
C04920=1025.279,388.867,352.408,172.918,48.620,159.774
C04921=1025.270,388.620,352.451,172.908,48.619,159.773
C04922=1025.261,388.374,352.493,172.899,48.618,159.771
C04923=1025.252,388.128,352.536,172.890,48.616,159.769
C04924=1025.242,387.881,352.579,172.880,48.615,159.767
C04925=1025.233,387.636,352.621,172.871,48.614,159.765
C04926=1025.224,387.390,352.664,172.860,48.613,159.764
C04927=1025.214,387.143,352.706,172.851,48.611,159.762
C04928=1025.205,386.897,352.748,172.842,48.609,159.760
C04929=1025.196,386.651,352.791,172.833,48.608,159.758
C04930=1025.188,386.405,352.833,172.823,48.607,159.757
C04931=1025.178,386.158,352.876,172.814,48.605,159.755
C04932=1025.169,385.912,352.917,172.804,48.604,159.753
C04933=1025.160,385.666,352.960,172.794,48.603,159.751
C04934=1025.151,385.420,353.002,172.785,48.602,159.750
C04935=1025.141,385.174,353.044,172.776,48.600,159.748
C04936=1025.132,384.927,353.086,172.767,48.599,159.746
C04937=1025.122,384.681,353.127,172.757,48.598,159.745
C04938=1025.113,384.435,353.169,172.748,48.596,159.743
C04939=1025.104,384.189,353.211,172.739,48.596,159.741
C04940=1025.095,383.943,353.253,172.730,48.594,159.740
C04941=1025.086,383.696,353.295,172.721,48.593,159.738
C04942=1025.077,383.450,353.337,172.711,48.592,159.736
C04943=1025.068,383.203,353.378,172.702,48.591,159.735
C04944=1025.059,382.957,353.420,172.693,48.590,159.733
C04945=1025.050,382.711,353.462,172.684,48.588,159.731
C04946=1025.041,382.465,353.504,172.675,48.587,159.730
C04947=1025.032,382.219,353.546,172.666,48.586,159.728
C04948=1025.023,381.973,353.587,172.657,48.585,159.727
C04949=1025.014,381.726,353.629,172.647,48.584,159.725
C04950=1025.005,381.479,353.670,172.638,48.583,159.723
C04951=1024.992,381.127,353.729,172.626,48.582,159.721
C04952=1024.980,380.775,353.789,172.613,48.580,159.719
C04953=1024.967,380.422,353.848,172.600,48.578,159.716
C04954=1024.955,380.071,353.908,172.588,48.577,159.714
C04955=1024.946,379.824,353.949,172.578,48.576,159.713
C04956=1024.937,379.577,353.990,172.570,48.575,159.711
C04957=1024.928,379.331,354.032,172.561,48.574,159.710
C04958=1024.919,379.085,354.072,172.552,48.573,159.708
C04959=1024.910,378.839,354.114,172.543,48.572,159.707
C04960=1024.902,378.592,354.155,172.534,48.571,159.705
C04961=1024.893,378.345,354.197,172.526,48.570,159.704
C04962=1024.884,378.100,354.238,172.517,48.570,159.702
C04963=1024.876,377.853,354.279,172.508,48.569,159.701
C04964=1024.867,377.606,354.321,172.499,48.568,159.699
C04965=1024.859,377.360,354.361,172.492,48.567,159.698
C04966=1024.850,377.113,354.402,172.482,48.565,159.696
C04967=1024.842,376.867,354.444,172.474,48.565,159.694
C04968=1024.833,376.621,354.484,172.465,48.564,159.693
C04969=1024.824,376.374,354.525,172.457,48.564,159.692
C04970=1024.815,376.128,354.565,172.448,48.563,159.690
C04971=1024.807,375.881,354.606,172.439,48.562,159.689
C04972=1024.798,375.634,354.647,172.430,48.561,159.687
C04973=1024.789,375.388,354.688,172.422,48.560,159.686
C04974=1024.780,375.141,354.729,172.414,48.560,159.684
C04975=1024.771,374.895,354.769,172.405,48.559,159.683
C04976=1024.763,374.648,354.810,172.397,48.558,159.681
C04977=1024.754,374.402,354.850,172.388,48.558,159.680
C04978=1024.746,374.155,354.890,172.379,48.557,159.679
C04979=1024.737,373.909,354.930,172.371,48.556,159.677
C04980=1024.728,373.662,354.971,172.363,48.556,159.676
C04981=1024.720,373.416,355.012,172.355,48.555,159.674
C04982=1024.712,373.170,355.052,172.346,48.555,159.673
C04983=1024.703,372.923,355.093,172.337,48.554,159.672
C04984=1024.694,372.676,355.132,172.330,48.553,159.670
C04985=1024.686,372.429,355.173,172.321,48.552,159.669
C04986=1024.677,372.183,355.213,172.313,48.552,159.668
C04987=1024.669,371.937,355.254,172.304,48.551,159.666
C04988=1024.660,371.690,355.294,172.297,48.551,159.665
C04989=1024.652,371.443,355.334,172.288,48.550,159.663
C04990=1024.643,371.197,355.374,172.280,48.550,159.662
C04991=1024.635,370.950,355.415,172.271,48.549,159.661
C04992=1024.627,370.703,355.455,172.263,48.548,159.659
C04993=1024.618,370.457,355.495,172.255,48.548,159.658
C04994=1024.610,370.210,355.535,172.247,48.548,159.657
C04995=1024.602,369.964,355.574,172.239,48.547,159.656
C04996=1024.594,369.716,355.615,172.230,48.546,159.654
C04997=1024.585,369.470,355.655,172.223,48.546,159.653
C04998=1024.577,369.223,355.695,172.215,48.546,159.652
C04999=1024.568,368.977,355.735,172.206,48.545,159.650
C05000=1024.561,368.731,355.775,172.199,48.545,159.649
C05001=1024.552,368.484,355.814,172.190,48.544,159.648
C05002=1024.544,368.236,355.854,172.182,48.544,159.646
C05003=1024.535,367.990,355.894,172.175,48.544,159.645
C05004=1024.527,367.744,355.934,172.166,48.543,159.644
C05005=1024.518,367.497,355.973,172.159,48.543,159.643
C05006=1024.510,367.250,356.013,172.150,48.543,159.641
C05007=1024.502,367.016,356.050,172.143,48.542,159.640
C05008=1024.494,366.783,356.088,172.135,48.542,159.639
C05009=1024.487,366.549,356.124,172.128,48.542,159.638
C05010=1024.478,366.316,356.162,172.120,48.541,159.637
C05011=1024.470,366.082,356.199,172.113,48.541,159.636
C05012=1024.463,365.848,356.237,172.106,48.541,159.634
C05013=1024.455,365.614,356.274,172.097,48.540,159.633
C05014=1024.447,365.381,356.311,172.090,48.541,159.632
C05015=1024.439,365.134,356.350,172.083,48.540,159.631
C05016=1024.430,364.887,356.389,172.074,48.540,159.630
C05017=1024.423,364.640,356.429,172.067,48.540,159.629
C05018=1024.414,364.393,356.469,172.059,48.539,159.627
C05019=1024.406,364.146,356.507,172.052,48.540,159.626
C05020=1024.398,363.900,356.547,172.044,48.539,159.625
C05021=1024.390,363.654,356.586,172.036,48.539,159.624
C05022=1024.382,363.406,356.625,172.028,48.539,159.623
C05023=1024.374,363.160,356.664,172.021,48.538,159.621
C05024=1024.365,362.913,356.703,172.013,48.539,159.620
C05025=1024.357,362.666,356.742,172.005,48.538,159.619
C05026=1024.349,362.419,356.781,171.997,48.539,159.618
C05027=1024.342,362.172,356.820,171.990,48.538,159.617
C05028=1024.334,361.926,356.859,171.983,48.538,159.616
C05029=1024.325,361.679,356.898,171.974,48.538,159.615
C05030=1024.317,361.432,356.937,171.967,48.538,159.613
C05031=1024.309,361.186,356.976,171.959,48.538,159.612
C05032=1024.302,360.939,357.016,171.952,48.538,159.611
C05033=1024.294,360.691,357.054,171.945,48.538,159.610
C05034=1024.285,360.444,357.093,171.937,48.538,159.609
C05035=1024.278,360.198,357.132,171.929,48.537,159.608
C05036=1024.269,359.951,357.170,171.922,48.537,159.607
C05037=1024.261,359.704,357.209,171.914,48.538,159.606
C05038=1024.254,359.457,357.247,171.907,48.538,159.605
C05039=1024.246,359.210,357.286,171.899,48.538,159.604
C05040=1024.237,358.963,357.324,171.892,48.538,159.603
C05041=1024.230,358.716,357.363,171.885,48.537,159.601
C05042=1024.222,358.469,357.401,171.877,48.538,159.600
C05043=1024.214,358.223,357.439,171.869,48.538,159.599
C05044=1024.206,357.975,357.478,171.862,48.538,159.598
C05045=1024.197,357.729,357.516,171.854,48.538,159.597
C05046=1024.190,357.482,357.554,171.847,48.538,159.596
C05047=1024.181,357.235,357.593,171.840,48.538,159.595
C05048=1024.174,356.988,357.631,171.832,48.539,159.594
C05049=1024.166,356.741,357.670,171.825,48.539,159.593
C05050=1024.158,356.495,357.708,171.818,48.539,159.592
C05051=1024.150,356.247,357.747,171.811,48.539,159.591
C05052=1024.143,356.000,357.784,171.803,48.540,159.590
C05053=1024.134,355.753,357.822,171.796,48.540,159.589
C05054=1024.126,355.507,357.860,171.789,48.540,159.588
C05055=1024.118,355.260,357.899,171.781,48.540,159.587
C05056=1024.111,355.012,357.937,171.774,48.541,159.586
C05057=1024.103,354.765,357.975,171.767,48.541,159.585
C05058=1024.095,354.519,358.013,171.760,48.541,159.584
C05059=1024.087,354.271,358.051,171.753,48.541,159.583
C05060=1024.079,354.025,358.089,171.746,48.542,159.582
C05061=1024.072,353.778,358.127,171.738,48.542,159.581
C05062=1024.063,353.531,358.165,171.732,48.542,159.580
C05063=1024.056,353.284,358.202,171.725,48.542,159.579
C05064=1024.048,353.036,358.241,171.717,48.543,159.578
C05065=1024.040,352.789,358.278,171.710,48.543,159.577
C05066=1024.032,352.542,358.315,171.703,48.543,159.576
C05067=1024.025,352.312,358.350,171.696,48.544,159.575
C05068=1024.018,352.082,358.386,171.689,48.544,159.575
C05069=1024.010,351.851,358.421,171.683,48.544,159.574
C05070=1024.003,351.621,358.456,171.677,48.545,159.573
C05071=1023.995,351.391,358.491,171.670,48.545,159.572
C05072=1023.989,351.160,358.526,171.663,48.545,159.571
C05073=1023.982,350.930,358.561,171.657,48.546,159.570
C05074=1023.974,350.700,358.596,171.650,48.546,159.569
C05075=1023.967,350.453,358.634,171.644,48.547,159.568
C05076=1023.959,350.206,358.671,171.637,48.547,159.567
C05077=1023.951,349.958,358.709,171.629,48.548,159.567
C05078=1023.944,349.711,358.746,171.622,48.549,159.566
C05079=1023.936,349.465,358.784,171.615,48.549,159.565
C05080=1023.929,349.218,358.821,171.608,48.549,159.564
C05081=1023.921,348.971,358.859,171.602,48.550,159.563
C05082=1023.913,348.724,358.896,171.595,48.550,159.562
C05083=1023.905,348.476,358.934,171.588,48.550,159.561
C05084=1023.898,348.229,358.971,171.581,48.551,159.560
C05085=1023.890,347.982,359.008,171.575,48.552,159.560
C05086=1023.883,347.734,359.045,171.567,48.553,159.559
C05087=1023.875,347.488,359.082,171.560,48.553,159.558
C05088=1023.868,347.240,359.119,171.553,48.554,159.557
C05089=1023.860,346.994,359.156,171.547,48.555,159.556
C05090=1023.852,346.747,359.193,171.540,48.555,159.555
C05091=1023.845,346.499,359.230,171.533,48.556,159.554
C05092=1023.837,346.252,359.267,171.527,48.556,159.554
C05093=1023.830,346.005,359.305,171.520,48.557,159.553
C05094=1023.822,345.758,359.341,171.513,48.558,159.552
C05095=1023.814,345.511,359.378,171.506,48.558,159.551
C05096=1023.807,345.264,359.415,171.500,48.559,159.550
C05097=1023.799,345.016,359.451,171.493,48.559,159.549
C05098=1023.792,344.769,359.489,171.486,48.560,159.549
C05099=1023.784,344.522,359.526,171.480,48.561,159.548
C05100=1023.776,344.275,359.562,171.473,48.561,159.547
C05101=1023.769,344.028,359.600,171.466,48.562,159.546
C05102=1023.762,343.780,359.636,171.460,48.563,159.546
C05103=1023.754,343.533,359.673,171.453,48.564,159.545
C05104=1023.747,343.286,359.710,171.446,48.564,159.544
C05105=1023.739,343.038,359.746,171.440,48.565,159.543
C05106=1023.731,342.791,359.783,171.433,48.566,159.542
C05107=1023.725,342.544,359.819,171.426,48.567,159.542
C05108=1023.717,342.297,359.856,171.420,48.568,159.541
C05109=1023.709,342.050,359.892,171.413,48.568,159.540
C05110=1023.702,341.802,359.929,171.407,48.569,159.539
C05111=1023.694,341.555,359.966,171.400,48.570,159.538
C05112=1023.687,341.309,360.002,171.394,48.571,159.538
C05113=1023.680,341.061,360.039,171.387,48.572,159.537
C05114=1023.672,340.813,360.075,171.380,48.572,159.536
C05115=1023.665,340.566,360.111,171.374,48.574,159.535
C05116=1023.657,340.320,360.148,171.367,48.574,159.535
C05117=1023.650,340.072,360.185,171.361,48.576,159.534
C05118=1023.643,339.825,360.221,171.354,48.576,159.533
C05119=1023.635,339.577,360.257,171.348,48.577,159.533
C05120=1023.628,339.331,360.293,171.341,48.578,159.532
C05121=1023.620,339.083,360.329,171.335,48.579,159.531
C05122=1023.613,338.836,360.365,171.328,48.580,159.530
C05123=1023.605,338.588,360.401,171.321,48.581,159.530
C05124=1023.598,338.341,360.437,171.315,48.582,159.529
C05125=1023.590,338.094,360.474,171.308,48.583,159.528
C05126=1023.583,337.846,360.510,171.302,48.584,159.527
C05127=1023.577,337.614,360.543,171.297,48.585,159.527
C05128=1023.569,337.382,360.577,171.290,48.586,159.526
C05129=1023.563,337.151,360.611,171.285,48.587,159.526
C05130=1023.555,336.919,360.645,171.278,48.588,159.525
C05131=1023.549,336.687,360.678,171.273,48.589,159.524
C05132=1023.541,336.455,360.712,171.266,48.590,159.524
C05133=1023.535,336.224,360.746,171.261,48.591,159.523
C05134=1023.528,335.992,360.780,171.255,48.592,159.522
C05135=1023.521,335.744,360.815,171.248,48.593,159.522
C05136=1023.513,335.497,360.851,171.242,48.594,159.521
C05137=1023.506,335.250,360.887,171.235,48.595,159.520
C05138=1023.499,335.002,360.922,171.230,48.596,159.520
C05139=1023.492,334.755,360.958,171.223,48.597,159.519
C05140=1023.484,334.508,360.995,171.217,48.599,159.519
C05141=1023.477,334.260,361.030,171.211,48.600,159.518
C05142=1023.470,334.013,361.066,171.204,48.601,159.517
C05143=1023.463,333.766,361.101,171.198,48.602,159.517
C05144=1023.455,333.518,361.137,171.193,48.603,159.516
C05145=1023.449,333.271,361.172,171.186,48.605,159.515
C05146=1023.441,333.023,361.209,171.180,48.606,159.515
C05147=1023.434,332.776,361.244,171.173,48.607,159.514
C05148=1023.427,332.529,361.279,171.167,48.608,159.513
C05149=1023.419,332.281,361.315,171.161,48.609,159.513
C05150=1023.412,332.034,361.350,171.154,48.611,159.512
C05151=1023.405,331.786,361.385,171.149,48.612,159.512
C05152=1023.398,331.539,361.421,171.143,48.613,159.511
C05153=1023.390,331.292,361.456,171.137,48.615,159.511
C05154=1023.383,331.044,361.491,171.130,48.616,159.510
C05155=1023.376,330.797,361.526,171.124,48.617,159.509
C05156=1023.368,330.549,361.562,171.118,48.618,159.509
C05157=1023.362,330.302,361.598,171.112,48.620,159.508
C05158=1023.354,330.055,361.632,171.106,48.621,159.508
C05159=1023.347,329.808,361.667,171.100,48.622,159.507
C05160=1023.340,329.560,361.703,171.093,48.624,159.506
C05161=1023.333,329.312,361.738,171.088,48.625,159.506
C05162=1023.326,329.065,361.772,171.082,48.626,159.505
C05163=1023.318,328.818,361.809,171.075,48.628,159.505
C05164=1023.311,328.570,361.844,171.069,48.630,159.504
C05165=1023.305,328.323,361.879,171.063,48.631,159.504
C05166=1023.297,328.076,361.913,171.058,48.632,159.503
C05167=1023.290,327.828,361.949,171.052,48.634,159.503
C05168=1023.283,327.580,361.984,171.045,48.635,159.502
C05169=1023.276,327.333,362.019,171.039,48.637,159.501
C05170=1023.269,327.086,362.054,171.034,48.638,159.501
C05171=1023.262,326.838,362.088,171.028,48.639,159.500
C05172=1023.255,326.591,362.123,171.021,48.641,159.500
C05173=1023.247,326.343,362.158,171.015,48.643,159.499
C05174=1023.240,326.096,362.193,171.009,48.644,159.499
C05175=1023.233,325.848,362.227,171.004,48.645,159.498
C05176=1023.226,325.601,362.262,170.998,48.647,159.498
C05177=1023.218,325.354,362.296,170.992,48.648,159.497
C05178=1023.211,325.105,362.330,170.986,48.650,159.497
C05179=1023.204,324.858,362.366,170.979,48.652,159.496
C05180=1023.196,324.611,362.400,170.974,48.654,159.496
C05181=1023.189,324.363,362.434,170.968,48.655,159.495
C05182=1023.182,324.116,362.469,170.962,48.657,159.495
C05183=1023.175,323.868,362.503,170.956,48.659,159.494
C05184=1023.168,323.621,362.537,170.951,48.660,159.494
C05185=1023.161,323.373,362.572,170.945,48.661,159.493
C05186=1023.154,323.126,362.606,170.939,48.663,159.493
C05187=1023.147,322.892,362.639,170.934,48.665,159.493
C05188=1023.139,322.658,362.671,170.928,48.667,159.492
C05189=1023.133,322.423,362.704,170.922,48.668,159.492
C05190=1023.126,322.189,362.736,170.916,48.670,159.491
C05191=1023.120,321.956,362.769,170.911,48.671,159.491
C05192=1023.113,321.721,362.801,170.906,48.673,159.490
C05193=1023.107,321.487,362.833,170.900,48.674,159.490
C05194=1023.099,321.253,362.866,170.895,48.676,159.489
C05195=1023.092,321.005,362.900,170.889,48.678,159.489
C05196=1023.086,320.757,362.934,170.883,48.680,159.489
C05197=1023.078,320.510,362.969,170.878,48.681,159.488
C05198=1023.071,320.262,363.003,170.872,48.683,159.488
C05199=1023.064,320.015,363.037,170.866,48.685,159.487
C05200=1023.058,319.768,363.071,170.861,48.687,159.487
C05201=1023.051,319.520,363.105,170.855,48.688,159.486
C05202=1023.043,319.273,363.139,170.849,48.690,159.486
C05203=1023.037,319.025,363.173,170.844,48.692,159.486
C05204=1023.030,318.777,363.207,170.838,48.694,159.485
C05205=1023.022,318.530,363.242,170.832,48.696,159.485
C05206=1023.016,318.282,363.276,170.827,48.697,159.484
C05207=1023.009,318.035,363.310,170.821,48.699,159.484
C05208=1023.002,317.787,363.343,170.814,48.701,159.483
C05209=1022.995,317.540,363.377,170.810,48.703,159.483
C05210=1022.988,317.292,363.412,170.804,48.705,159.483
C05211=1022.981,317.044,363.446,170.798,48.707,159.482
C05212=1022.974,316.797,363.479,170.793,48.708,159.482
C05213=1022.968,316.549,363.513,170.787,48.710,159.481
C05214=1022.961,316.302,363.547,170.781,48.712,159.481
C05215=1022.954,316.054,363.581,170.776,48.714,159.481
C05216=1022.947,315.807,363.615,170.770,48.716,159.480
C05217=1022.941,315.559,363.649,170.765,48.718,159.480
C05218=1022.933,315.311,363.683,170.759,48.719,159.480
C05219=1022.927,315.064,363.716,170.753,48.721,159.479
C05220=1022.920,314.816,363.751,170.748,48.724,159.479
C05221=1022.913,314.569,363.784,170.742,48.725,159.478
C05222=1022.906,314.322,363.818,170.736,48.727,159.478
C05223=1022.899,314.074,363.852,170.731,48.729,159.478
C05224=1022.893,313.826,363.886,170.725,48.731,159.477
C05225=1022.887,313.578,363.919,170.720,48.733,159.477
C05226=1022.879,313.331,363.953,170.715,48.735,159.477
C05227=1022.872,313.083,363.987,170.710,48.737,159.476
C05228=1022.866,312.836,364.021,170.703,48.739,159.476
C05229=1022.859,312.588,364.054,170.698,48.741,159.476
C05230=1022.853,312.340,364.087,170.693,48.743,159.475
C05231=1022.846,312.092,364.122,170.687,48.745,159.475
C05232=1022.840,311.845,364.155,170.682,48.747,159.475
C05233=1022.832,311.598,364.189,170.676,48.749,159.474
C05234=1022.826,311.350,364.222,170.671,48.751,159.474
C05235=1022.820,311.102,364.256,170.665,48.753,159.473
C05236=1022.813,310.855,364.289,170.660,48.755,159.473
C05237=1022.806,310.607,364.323,170.655,48.757,159.473
C05238=1022.800,310.360,364.356,170.649,48.759,159.473
C05239=1022.793,310.112,364.389,170.644,48.761,159.472
C05240=1022.786,309.865,364.423,170.638,48.763,159.472
C05241=1022.779,309.617,364.455,170.632,48.766,159.472
C05242=1022.772,309.370,364.489,170.628,48.768,159.471
C05243=1022.765,309.121,364.522,170.622,48.770,159.471
C05244=1022.758,308.874,364.554,170.617,48.772,159.471
C05245=1022.751,308.626,364.587,170.611,48.775,159.471
C05246=1022.744,308.379,364.620,170.606,48.777,159.470
C05247=1022.738,308.147,364.650,170.601,48.779,159.470
C05248=1022.731,307.916,364.682,170.596,48.781,159.470
C05249=1022.724,307.684,364.712,170.591,48.783,159.469
C05250=1022.718,307.452,364.743,170.586,48.786,159.469
C05251=1022.712,307.221,364.774,170.581,48.788,159.469
C05252=1022.705,306.989,364.804,170.576,48.790,159.469
C05253=1022.699,306.757,364.835,170.571,48.792,159.468
C05254=1022.692,306.526,364.866,170.565,48.794,159.468
C05255=1022.686,306.279,364.898,170.561,48.796,159.468
C05256=1022.679,306.030,364.931,170.555,48.799,159.468
C05257=1022.672,305.783,364.964,170.550,48.801,159.468
C05258=1022.665,305.536,364.996,170.545,48.804,159.467
C05259=1022.658,305.288,365.029,170.539,48.806,159.467
C05260=1022.652,305.040,365.062,170.534,48.808,159.467
C05261=1022.645,304.792,365.095,170.529,48.811,159.467
C05262=1022.638,304.544,365.127,170.524,48.813,159.466
C05263=1022.631,304.297,365.160,170.518,48.815,159.466
C05264=1022.624,304.048,365.193,170.514,48.818,159.466
C05265=1022.617,303.801,365.225,170.508,48.820,159.466
C05266=1022.611,303.554,365.258,170.502,48.823,159.465
C05267=1022.603,303.306,365.290,170.497,48.825,159.465
C05268=1022.597,303.058,365.323,170.492,48.827,159.465
C05269=1022.591,302.810,365.356,170.487,48.830,159.465
C05270=1022.584,302.563,365.388,170.481,48.832,159.464
C05271=1022.577,302.314,365.420,170.477,48.835,159.464
C05272=1022.571,302.067,365.453,170.471,48.837,159.464
C05273=1022.564,301.819,365.485,170.467,48.840,159.464
C05274=1022.558,301.572,365.518,170.461,48.842,159.464
C05275=1022.550,301.324,365.550,170.456,48.844,159.463
C05276=1022.544,301.076,365.583,170.451,48.847,159.463
C05277=1022.538,300.828,365.615,170.445,48.850,159.463
C05278=1022.531,300.581,365.647,170.441,48.852,159.463
C05279=1022.524,300.333,365.680,170.435,48.855,159.463
C05280=1022.517,300.085,365.712,170.430,48.857,159.462
C05281=1022.511,299.837,365.744,170.424,48.859,159.462
C05282=1022.505,299.589,365.777,170.420,48.862,159.462
C05283=1022.497,299.342,365.809,170.414,48.865,159.462
C05284=1022.492,299.094,365.841,170.410,48.867,159.462
C05285=1022.484,298.847,365.874,170.404,48.869,159.461
C05286=1022.478,298.598,365.907,170.400,48.872,159.461
C05287=1022.472,298.350,365.939,170.394,48.875,159.461
C05288=1022.465,298.103,365.971,170.389,48.877,159.461
C05289=1022.459,297.855,366.003,170.384,48.880,159.461
C05290=1022.452,297.607,366.035,170.379,48.882,159.461
C05291=1022.446,297.359,366.067,170.374,48.885,159.460
C05292=1022.439,297.111,366.100,170.369,48.888,159.460
C05293=1022.432,296.864,366.132,170.364,48.890,159.460
C05294=1022.426,296.616,366.164,170.359,48.893,159.460
C05295=1022.419,296.369,366.196,170.355,48.895,159.460
C05296=1022.413,296.120,366.228,170.349,48.898,159.460
C05297=1022.407,295.872,366.260,170.344,48.901,159.460
C05298=1022.400,295.625,366.292,170.339,48.903,159.459
C05299=1022.394,295.377,366.324,170.334,48.906,159.459
C05300=1022.387,295.129,366.356,170.329,48.909,159.459
C05301=1022.381,294.881,366.388,170.324,48.911,159.459
C05302=1022.375,294.634,366.421,170.319,48.914,159.459
C05303=1022.368,294.386,366.453,170.314,48.917,159.459
C05304=1022.362,294.138,366.485,170.309,48.919,159.459
C05305=1022.355,293.890,366.517,170.304,48.922,159.459
C05306=1022.349,293.642,366.549,170.300,48.924,159.458
C05307=1022.343,293.419,366.577,170.295,48.927,159.458
C05308=1022.337,293.197,366.606,170.291,48.929,159.458
C05309=1022.332,292.973,366.634,170.286,48.932,159.458
C05310=1022.326,292.751,366.663,170.282,48.934,159.458
C05311=1022.320,292.528,366.692,170.277,48.937,159.458
C05312=1022.314,292.305,366.720,170.273,48.940,159.458
C05313=1022.308,292.082,366.749,170.268,48.942,159.458
C05314=1022.303,291.860,366.777,170.264,48.945,159.457
C05315=1022.296,291.612,366.808,170.259,48.947,159.457
C05316=1022.289,291.364,366.840,170.254,48.951,159.457
C05317=1022.283,291.116,366.871,170.249,48.953,159.457
C05318=1022.276,290.868,366.903,170.244,48.956,159.457
C05319=1022.269,290.620,366.934,170.240,48.959,159.457
C05320=1022.262,290.372,366.965,170.234,48.962,159.457
C05321=1022.256,290.124,366.997,170.230,48.965,159.457
C05322=1022.250,289.876,367.029,170.224,48.968,159.457
C05323=1022.243,289.628,367.060,170.220,48.971,159.457
C05324=1022.236,289.380,367.092,170.214,48.973,159.457
C05325=1022.230,289.133,367.122,170.210,48.976,159.457
C05326=1022.224,288.885,367.154,170.205,48.979,159.457
C05327=1022.217,288.637,367.185,170.200,48.982,159.457
C05328=1022.210,288.389,367.216,170.195,48.986,159.456
C05329=1022.203,288.141,367.248,170.191,48.988,159.456
C05330=1022.198,287.893,367.280,170.185,48.992,159.456
C05331=1022.192,287.645,367.310,170.181,48.994,159.456
C05332=1022.185,287.397,367.342,170.176,48.998,159.456
C05333=1022.178,287.149,367.373,170.171,49.000,159.456
C05334=1022.172,286.901,367.405,170.166,49.004,159.456
C05335=1022.166,286.653,367.435,170.162,49.006,159.456
C05336=1022.159,286.405,367.466,170.156,49.010,159.456
C05337=1022.152,286.158,367.498,170.152,49.012,159.456
C05338=1022.146,285.909,367.528,170.147,49.016,159.456
C05339=1022.139,285.661,367.560,170.142,49.019,159.456
C05340=1022.133,285.414,367.591,170.138,49.021,159.456
C05341=1022.127,285.165,367.622,170.133,49.025,159.456
C05342=1022.120,284.918,367.653,170.129,49.028,159.456
C05343=1022.113,284.670,367.683,170.123,49.031,159.456
C05344=1022.107,284.422,367.714,170.119,49.034,159.456
C05345=1022.100,284.174,367.745,170.114,49.037,159.456
C05346=1022.093,283.926,367.776,170.109,49.040,159.456
C05347=1022.088,283.678,367.807,170.104,49.044,159.456
C05348=1022.081,283.430,367.838,170.100,49.047,159.456
C05349=1022.074,283.182,367.868,170.095,49.050,159.456
C05350=1022.067,282.934,367.900,170.091,49.054,159.456
C05351=1022.061,282.686,367.930,170.085,49.057,159.456
C05352=1022.055,282.437,367.961,170.081,49.060,159.456
C05353=1022.048,282.190,367.992,170.076,49.063,159.456
C05354=1022.041,281.942,368.022,170.072,49.066,159.456
C05355=1022.035,281.694,368.053,170.066,49.069,159.456
C05356=1022.028,281.446,368.084,170.062,49.072,159.456
C05357=1022.023,281.198,368.115,170.057,49.076,159.456
C05358=1022.016,280.949,368.145,170.053,49.079,159.456
C05359=1022.009,280.702,368.176,170.047,49.082,159.456
C05360=1022.003,280.454,368.206,170.043,49.086,159.456
C05361=1021.996,280.205,368.237,170.039,49.089,159.456
C05362=1021.991,279.958,368.267,170.034,49.092,159.456
C05363=1021.984,279.710,368.299,170.030,49.095,159.456
C05364=1021.977,279.462,368.329,170.024,49.099,159.456
C05365=1021.971,279.214,368.359,170.020,49.102,159.456
C05366=1021.965,278.966,368.390,170.015,49.105,159.456
C05367=1021.959,278.749,368.417,170.011,49.108,159.456
C05368=1021.953,278.533,368.443,170.008,49.111,159.456
C05369=1021.948,278.315,368.471,170.003,49.114,159.456
C05370=1021.942,278.099,368.497,169.999,49.117,159.456
C05371=1021.937,277.882,368.523,169.995,49.120,159.456
C05372=1021.931,277.665,368.550,169.991,49.122,159.456
C05373=1021.926,277.449,368.577,169.987,49.126,159.457
C05374=1021.921,277.232,368.604,169.983,49.129,159.457
C05375=1021.914,276.984,368.634,169.979,49.132,159.457
C05376=1021.908,276.736,368.664,169.974,49.136,159.457
C05377=1021.901,276.488,368.694,169.969,49.138,159.457
C05378=1021.895,276.240,368.725,169.964,49.142,159.457
C05379=1021.888,275.992,368.756,169.960,49.146,159.457
C05380=1021.882,275.744,368.785,169.955,49.149,159.457
C05381=1021.876,275.495,368.815,169.951,49.153,159.457
C05382=1021.869,275.247,368.845,169.946,49.156,159.457
C05383=1021.863,275.000,368.875,169.942,49.160,159.457
C05384=1021.856,274.751,368.906,169.938,49.163,159.457
C05385=1021.850,274.504,368.936,169.933,49.167,159.457
C05386=1021.843,274.255,368.966,169.929,49.170,159.457
C05387=1021.837,274.008,368.996,169.923,49.173,159.457
C05388=1021.831,273.759,369.026,169.919,49.177,159.458
C05389=1021.825,273.511,369.056,169.914,49.181,159.458
C05390=1021.818,273.263,369.086,169.910,49.184,159.458
C05391=1021.812,273.015,369.117,169.905,49.187,159.458
C05392=1021.806,272.767,369.147,169.901,49.191,159.458
C05393=1021.799,272.518,369.176,169.896,49.195,159.458
C05394=1021.793,272.271,369.206,169.892,49.198,159.458
C05395=1021.786,272.022,369.237,169.887,49.202,159.458
C05396=1021.780,271.774,369.266,169.883,49.206,159.458
C05397=1021.774,271.526,369.296,169.879,49.209,159.459
C05398=1021.767,271.278,369.326,169.874,49.213,159.459
C05399=1021.761,271.030,369.356,169.870,49.216,159.459
C05400=1021.755,270.782,369.386,169.865,49.220,159.459
C05401=1021.748,270.533,369.416,169.861,49.223,159.459
C05402=1021.742,270.285,369.445,169.856,49.227,159.459
C05403=1021.736,270.038,369.475,169.852,49.231,159.459
C05404=1021.729,269.789,369.505,169.847,49.235,159.459
C05405=1021.723,269.541,369.535,169.843,49.238,159.460
C05406=1021.717,269.293,369.565,169.838,49.242,159.460
C05407=1021.710,269.045,369.595,169.834,49.246,159.460
C05408=1021.704,268.796,369.624,169.829,49.250,159.460
C05409=1021.697,268.549,369.654,169.825,49.253,159.460
C05410=1021.692,268.300,369.683,169.821,49.257,159.460
C05411=1021.685,268.052,369.713,169.816,49.260,159.460
C05412=1021.679,267.804,369.742,169.812,49.264,159.460
C05413=1021.673,267.556,369.773,169.807,49.268,159.461
C05414=1021.666,267.307,369.802,169.803,49.271,159.461
C05415=1021.660,267.059,369.831,169.799,49.276,159.461
C05416=1021.653,266.812,369.861,169.795,49.279,159.461
C05417=1021.648,266.563,369.891,169.790,49.283,159.461
C05418=1021.641,266.315,369.920,169.786,49.287,159.461
C05419=1021.634,266.067,369.950,169.781,49.291,159.462
C05420=1021.628,265.819,369.979,169.777,49.294,159.462
C05421=1021.622,265.570,370.008,169.772,49.298,159.462
C05422=1021.616,265.323,370.038,169.768,49.302,159.462
C05423=1021.609,265.074,370.068,169.763,49.306,159.462
C05424=1021.603,264.826,370.097,169.759,49.310,159.462
C05425=1021.596,264.578,370.126,169.754,49.314,159.463
C05426=1021.590,264.330,370.155,169.751,49.318,159.463
C05427=1021.585,264.116,370.181,169.747,49.321,159.463
C05428=1021.579,263.901,370.206,169.742,49.324,159.463
C05429=1021.573,263.686,370.231,169.739,49.328,159.463
C05430=1021.568,263.472,370.256,169.735,49.331,159.463
C05431=1021.563,263.258,370.282,169.731,49.335,159.464
C05432=1021.557,263.044,370.307,169.728,49.338,159.464
C05433=1021.552,262.829,370.332,169.724,49.341,159.464
C05434=1021.547,262.615,370.357,169.720,49.345,159.464
C05435=1021.541,262.366,370.386,169.716,49.349,159.464
C05436=1021.534,262.118,370.416,169.712,49.352,159.464
C05437=1021.528,261.869,370.445,169.708,49.357,159.465
C05438=1021.521,261.621,370.474,169.703,49.360,159.465
C05439=1021.515,261.373,370.503,169.699,49.365,159.465
C05440=1021.508,261.126,370.533,169.694,49.369,159.465
C05441=1021.503,260.877,370.562,169.690,49.372,159.466
C05442=1021.497,260.629,370.591,169.686,49.377,159.466
C05443=1021.490,260.381,370.620,169.682,49.380,159.466
C05444=1021.485,260.132,370.649,169.677,49.385,159.466
C05445=1021.478,259.884,370.677,169.673,49.388,159.466
C05446=1021.471,259.636,370.706,169.669,49.393,159.467
C05447=1021.464,259.387,370.735,169.665,49.397,159.467
C05448=1021.457,259.140,370.764,169.660,49.401,159.467
C05449=1021.452,258.891,370.792,169.656,49.405,159.468
C05450=1021.445,258.643,370.821,169.652,49.410,159.468
C05451=1021.438,258.395,370.850,169.647,49.414,159.468
C05452=1021.432,258.147,370.879,169.643,49.418,159.468
C05453=1021.426,257.898,370.907,169.639,49.422,159.469
C05454=1021.420,257.650,370.936,169.635,49.426,159.469
C05455=1021.413,257.402,370.965,169.630,49.430,159.469
